LIN {X 0,Y 369.299,Z 673.807,A -85,B 0,C 180,E1 -13026.444,E2 -13026.444} C_VEL
LIN {X 0,Y 367.685,Z 686.752,A -85,B 0,C 180,E1 -13027.673,E2 -13027.673} C_VEL
LIN {X 0,Y 366.094,Z 698.777,A -85,B 0,C 180,E1 -13029.05,E2 -13029.05} C_VEL
LIN {X 0,Y 364.688,Z 709.985,A -85,B 0,C 180,E1 -13030.584,E2 -13030.584} C_VEL
LIN {X 0,Y 363.393,Z 720.355,A -85,B 0,C 180,E1 -13032.266,E2 -13032.266} C_VEL
LIN {X 0,Y 362.264,Z 730.519,A -85,B 0,C 180,E1 -13034.24,E2 -13034.24} C_VEL
LIN {X 0,Y 361.681,Z 737.904,A -85,B 0,C 180,E1 -13035.943,E2 -13035.943} C_VEL
LIN {X 0,Y 361.141,Z 746.082,A -85,B 0,C 180,E1 -13038.209,E2 -13038.209} C_VEL
LIN {X 0,Y 361.017,Z 752.615,A -85,B 0,C 180,E1 -13040.475,E2 -13040.475} C_VEL
LIN {X 0,Y 361.096,Z 756.535,A -85,B 0,C 180,E1 -13042.169,E2 -13042.169} C_VEL
LIN {X 0,Y 361.282,Z 760.576,A -85,B 0,C 180,E1 -13044.418,E2 -13044.418} C_VEL
LIN {X 0,Y 361.402,Z 762.102,A -85,B 0,C 180,E1 -13045.538,E2 -13045.538} C_VEL
LIN {X 0,Y 361.443,Z 764.123,A -85,B 0,C 180,E1 -13047.771,E2 -13047.771} C_VEL
LIN {X 0,Y 361.687,Z 764.698,A -85,B 0,C 180,E1 -13048.886,E2 -13048.886} C_VEL
LIN {X 0,Y 361.681,Z 764.869,A -85,B 0,C 180,E1 -13051.113,E2 -13051.113} C_VEL
LIN {X 0,Y 361.357,Z 763.796,A -85,B 0,C 180,E1 -13053.344,E2 -13053.344} C_VEL
LIN {X 0,Y 361.354,Z 762.831,A -85,B 0,C 180,E1 -13054.461,E2 -13054.461} C_VEL
LIN {X 0,Y 361.099,Z 759.485,A -85,B 0,C 180,E1 -13056.975,E2 -13056.975} C_VEL
LIN {X 0,Y 360.902,Z 754.467,A -85,B 0,C 180,E1 -13059.527,E2 -13059.527} C_VEL
LIN {X 0,Y 361.06,Z 748.6,A -85,B 0,C 180,E1 -13061.793,E2 -13061.793} C_VEL
LIN {X 0,Y 361.615,Z 741.459,A -85,B 0,C 180,E1 -13064.002,E2 -13064.002} C_VEL
LIN {X 0,Y 362.603,Z 732.201,A -85,B 0,C 180,E1 -13066.321,E2 -13066.321} C_VEL
LIN {X 0,Y 363.986,Z 722.704,A -85,B 0,C 180,E1 -13068.285,E2 -13068.285} C_VEL
LIN {X 0,Y 365.41,Z 713.269,A -85,B 0,C 180,E1 -13069.931,E2 -13069.931} C_VEL
LIN {X 0,Y 367.365,Z 700.79,A -85,B 0,C 180,E1 -13071.755,E2 -13071.755} C_VEL
LIN {X 0,Y 369.396,Z 688.323,A -85,B 0,C 180,E1 -13073.251,E2 -13073.251} C_VEL
LIN {X 0,Y 371.558,Z 674.683,A -85,B 0,C 180,E1 -13074.589,E2 -13074.589} C_VEL
LIN {X 0,Y 373.499,Z 661.351,A -85,B 0,C 180,E1 -13075.643,E2 -13075.643} C_VEL
LIN {X 0,Y 375.455,Z 646.833,A -85,B 0,C 180,E1 -13076.544,E2 -13076.544} C_VEL
LIN {X 0,Y 377.1,Z 631.865,A -85,B 0,C 180,E1 -13077.242,E2 -13077.242} C_VEL
LIN {X 0,Y 378.235,Z 616.394,A -85,B 0,C 180,E1 -13077.753,E2 -13077.753} C_VEL
LIN {X 0,Y 379.231,Z 585.25,A -85,B 0,C 180,E1 -13078.389,E2 -13078.389} C_VEL
LIN {X 0,Y 381.27,Z 506.213,A -85,B 0,C 180,E1 -13079.919,E2 -13079.919} C_VEL
LIN {X 0,Y 378.126,Z 480.693,A -85,B 0,C 180,E1 -13080.781,E2 -13080.781} C_VEL
LIN {X 0,Y 373.205,Z 450.4,A -85,B 0,C 180,E1 -13081.959,E2 -13081.959} C_VEL
LIN {X 0,Y 372.138,Z 444.262,A -85,B 0,C 180,E1 -13082.225,E2 -13082.225} C_VEL
LIN {X 0,Y 374.167,Z 428.518,A -85,B 0,C 180,E1 -13084.622,E2 -13084.622} C_VEL
LIN {X 0,Y 371.816,Z 418.27,A -85,B 0,C 180,E1 -13086.551,E2 -13086.551} C_VEL
LIN {X 0,Y 367.323,Z 402.801,A -85,B 0,C 180,E1 -13089.726,E2 -13089.726} C_VEL
LIN {X 0,Y 362.493,Z 388.181,A -85,B 0,C 180,E1 -13093.024,E2 -13093.024} C_VEL
LIN {X 0,Y 361.834,Z 386.038,A -85,B 0,C 180,E1 -13093.563,E2 -13093.563} C_VEL
LIN {X 0,Y 361.819,Z 386.036,A -85,B 0,C 180,E1 -13097.169,E2 -13097.169} C_VEL
LIN {X 0,Y 361.815,Z 386.035,A -85,B 0,C 180,E1 -13100.982,E2 -13100.982} C_VEL
LIN {X 0,Y 361.859,Z 386.036,A -85,B 0,C 180,E1 -13104.656,E2 -13104.656} C_VEL
LIN {X 0,Y 361.827,Z 386.041,A -85,B 0,C 180,E1 -13108.37,E2 -13108.37} C_VEL
LIN {X 0,Y 361.855,Z 386.038,A -85,B 0,C 180,E1 -13110.952,E2 -13110.952} C_VEL
LIN {X 0,Y 361.84,Z 386.038,A -85,B 0,C 180,E1 -13114.704,E2 -13114.704} C_VEL
LIN {X 0,Y 361.84,Z 386.037,A -85,B 0,C 180,E1 -13118.344,E2 -13118.344} C_VEL
LIN {X 0,Y 361.883,Z 386.031,A -85,B 0,C 180,E1 -13122.097,E2 -13122.097} C_VEL
LIN {X 0,Y 361.968,Z 386.018,A -85,B 0,C 180,E1 -13126.113,E2 -13126.113} C_VEL
LIN {X 0,Y 361.984,Z 386.013,A -85,B 0,C 180,E1 -13129.937,E2 -13129.937} C_VEL
LIN {X 0,Y 362.102,Z 385.997,A -85,B 0,C 180,E1 -13133.313,E2 -13133.313} C_VEL
LIN {X 0,Y 362.254,Z 385.977,A -85,B 0,C 180,E1 -13137.777,E2 -13137.777} C_VEL
LIN {X 0,Y 362.252,Z 385.981,A -85,B 0,C 180,E1 -13142.224,E2 -13142.224} C_VEL
LIN {X 0,Y 362.127,Z 385.971,A -85,B 0,C 180,E1 -13146.687,E2 -13146.687} C_VEL
LIN {X 0,Y 361.985,Z 386.016,A -85,B 0,C 180,E1 -13150.064,E2 -13150.064} C_VEL
LIN {X 0,Y 361.987,Z 385.994,A -85,B 0,C 180,E1 -13153.899,E2 -13153.899} C_VEL
LIN {X 0,Y 361.917,Z 386.026,A -85,B 0,C 180,E1 -13156.935,E2 -13156.935} C_VEL
LIN {X 0,Y 361.873,Z 386.012,A -85,B 0,C 180,E1 -13160.462,E2 -13160.462} C_VEL
LIN {X 0,Y 361.851,Z 386.036,A -85,B 0,C 180,E1 -13164.102,E2 -13164.102} C_VEL
LIN {X 0,Y 361.826,Z 386.029,A -85,B 0,C 180,E1 -13167.786,E2 -13167.786} C_VEL
LIN {X 0,Y 361.837,Z 386.026,A -85,B 0,C 180,E1 -13171.286,E2 -13171.286} C_VEL
LIN {X 0,Y 361.842,Z 386.04,A -85,B 0,C 180,E1 -13174.282,E2 -13174.282} C_VEL
LIN {X 0,Y 361.851,Z 386.028,A -85,B 0,C 180,E1 -13177.223,E2 -13177.223} C_VEL
LIN {X 0,Y 361.805,Z 386.033,A -85,B 0,C 180,E1 -13180.752,E2 -13180.752} C_VEL
LIN {X 0,Y 361.806,Z 386.032,A -85,B 0,C 180,E1 -13184.371,E2 -13184.371} C_VEL
LIN {X 0,Y 361.822,Z 386.054,A -85,B 0,C 180,E1 -13188.265,E2 -13188.265} C_VEL
LIN {X 0,Y 362.805,Z 388.821,A -85,B 0,C 180,E1 -13188.449,E2 -13188.449} C_VEL
LIN {X 0,Y 364.536,Z 391.406,A -85,B 0,C 180,E1 -13188.714,E2 -13188.714} C_VEL
LIN {X 0,Y 374.281,Z 407.605,A -85,B 0,C 180,E1 -13190.185,E2 -13190.185} C_VEL
LIN {X 0,Y 382.972,Z 423.782,A -85,B 0,C 180,E1 -13191.447,E2 -13191.447} C_VEL
LIN {X 0,Y 381.952,Z 465.159,A -85,B 0,C 180,E1 -13192.26,E2 -13192.26} C_VEL
LIN {X 0,Y 380.904,Z 509.738,A -85,B 0,C 180,E1 -13193.136,E2 -13193.136} C_VEL
LIN {X 0,Y 380.569,Z 526.045,A -85,B 0,C 180,E1 -13193.572,E2 -13193.572} C_VEL
LIN {X 0,Y 379.947,Z 539.867,A -85,B 0,C 180,E1 -13194.138,E2 -13194.138} C_VEL
LIN {X 0,Y 378.941,Z 553.918,A -85,B 0,C 180,E1 -13194.906,E2 -13194.906} C_VEL
LIN {X 0,Y 377.652,Z 567.962,A -85,B 0,C 180,E1 -13195.903,E2 -13195.903} C_VEL
LIN {X 0,Y 376.21,Z 580.784,A -85,B 0,C 180,E1 -13197.039,E2 -13197.039} C_VEL
LIN {X 0,Y 374.328,Z 593.837,A -85,B 0,C 180,E1 -13198.444,E2 -13198.444} C_VEL
LIN {X 0,Y 372.539,Z 605.519,A -85,B 0,C 180,E1 -13199.987,E2 -13199.987} C_VEL
LIN {X 0,Y 370.658,Z 616.335,A -85,B 0,C 180,E1 -13201.706,E2 -13201.706} C_VEL
LIN {X 0,Y 368.828,Z 626.128,A -85,B 0,C 180,E1 -13203.584,E2 -13203.584} C_VEL
LIN {X 0,Y 367.11,Z 635.125,A -85,B 0,C 180,E1 -13205.696,E2 -13205.696} C_VEL
LIN {X 0,Y 365.859,Z 641.208,A -85,B 0,C 180,E1 -13207.408,E2 -13207.408} C_VEL
LIN {X 0,Y 364.601,Z 647.773,A -85,B 0,C 180,E1 -13209.699,E2 -13209.699} C_VEL
LIN {X 0,Y 363.547,Z 652.854,A -85,B 0,C 180,E1 -13211.983,E2 -13211.983} C_VEL
LIN {X 0,Y 362.813,Z 656.581,A -85,B 0,C 180,E1 -13214.266,E2 -13214.266} C_VEL
LIN {X 0,Y 362.312,Z 659.044,A -85,B 0,C 180,E1 -13216.541,E2 -13216.541} C_VEL
LIN {X 0,Y 362.042,Z 660.342,A -85,B 0,C 180,E1 -13218.807,E2 -13218.807} C_VEL
LIN {X 0,Y 361.94,Z 660.526,A -85,B 0,C 180,E1 -13221.064,E2 -13221.064} C_VEL
LIN {X 0,Y 362.002,Z 659.615,A -85,B 0,C 180,E1 -13223.311,E2 -13223.311} C_VEL
LIN {X 0,Y 362.04,Z 657.636,A -85,B 0,C 180,E1 -13225.547,E2 -13225.547} C_VEL
LIN {X 0,Y 362.519,Z 654.445,A -85,B 0,C 180,E1 -13227.778,E2 -13227.778} C_VEL
LIN {X 0,Y 362.987,Z 650.057,A -85,B 0,C 180,E1 -13230,E2 -13230} C_VEL
LIN {X 0,Y 363.879,Z 644.327,A -85,B 0,C 180,E1 -13232.214,E2 -13232.214} C_VEL
LIN {X 0,Y 364.903,Z 637.153,A -85,B 0,C 180,E1 -13234.419,E2 -13234.419} C_VEL
LIN {X 0,Y 365.957,Z 629.485,A -85,B 0,C 180,E1 -13236.34,E2 -13236.34} C_VEL
LIN {X 0,Y 367.335,Z 620.266,A -85,B 0,C 180,E1 -13238.25,E2 -13238.25} C_VEL
LIN {X 0,Y 368.656,Z 610.885,A -85,B 0,C 180,E1 -13239.88,E2 -13239.88} C_VEL
LIN {X 0,Y 370.067,Z 599.768,A -85,B 0,C 180,E1 -13241.502,E2 -13241.502} C_VEL
LIN {X 0,Y 371.296,Z 588.808,A -85,B 0,C 180,E1 -13242.851,E2 -13242.851} C_VEL
LIN {X 0,Y 372.593,Z 576.994,A -85,B 0,C 180,E1 -13244.055,E2 -13244.055} C_VEL
LIN {X 0,Y 373.78,Z 564.26,A -85,B 0,C 180,E1 -13245.123,E2 -13245.123} C_VEL
LIN {X 0,Y 374.814,Z 551.249,A -85,B 0,C 180,E1 -13245.999,E2 -13245.999} C_VEL
LIN {X 0,Y 374.608,Z 545.819,A -85,B 0,C 180,E1 -13246.354,E2 -13246.354} C_VEL
LIN {X 0,Y 372.444,Z 537.038,A -85,B 0,C 180,E1 -13246.98,E2 -13246.98} C_VEL
LIN {X 0,Y 370.164,Z 528.099,A -85,B 0,C 180,E1 -13247.538,E2 -13247.538} C_VEL
LIN {X 0,Y 369.641,Z 522.425,A -85,B 0,C 180,E1 -13247.777,E2 -13247.777} C_VEL
LIN {X 0,Y 369.882,Z 504.154,A -85,B 0,C 180,E1 -13248.217,E2 -13248.217} C_VEL
LIN {X 0,Y 371.608,Z 421.809,A -85,B 0,C 180,E1 -13249.832,E2 -13249.832} C_VEL
LIN {X 0,Y 359.643,Z 396.831,A -85,B 0,C 180,E1 -13251.356,E2 -13251.356} C_VEL
LIN {X 0,Y 355.091,Z 388.184,A -85,B 0,C 180,E1 -13251.946,E2 -13251.946} C_VEL
LIN {X 0,Y 354.805,Z 386.914,A -85,B 0,C 180,E1 -13252.006,E2 -13252.006} C_VEL
LIN {X 0,Y 354.795,Z 386.917,A -85,B 0,C 180,E1 -13255.835,E2 -13255.835} C_VEL
LIN {X 0,Y 354.786,Z 386.9,A -85,B 0,C 180,E1 -13259.684,E2 -13259.684} C_VEL
LIN {X 0,Y 354.786,Z 386.917,A -85,B 0,C 180,E1 -13262.333,E2 -13262.333} C_VEL
LIN {X 0,Y 354.817,Z 386.911,A -85,B 0,C 180,E1 -13265.697,E2 -13265.697} C_VEL
LIN {X 0,Y 354.767,Z 386.914,A -85,B 0,C 180,E1 -13269.412,E2 -13269.412} C_VEL
LIN {X 0,Y 354.764,Z 386.918,A -85,B 0,C 180,E1 -13272.862,E2 -13272.862} C_VEL
LIN {X 0,Y 354.756,Z 386.918,A -85,B 0,C 180,E1 -13276.101,E2 -13276.101} C_VEL
LIN {X 0,Y 354.76,Z 386.921,A -85,B 0,C 180,E1 -13279.175,E2 -13279.175} C_VEL
LIN {X 0,Y 354.795,Z 386.91,A -85,B 0,C 180,E1 -13282.404,E2 -13282.404} C_VEL
LIN {X 0,Y 354.804,Z 386.916,A -85,B 0,C 180,E1 -13284.939,E2 -13284.939} C_VEL
LIN {X 0,Y 354.771,Z 386.918,A -85,B 0,C 180,E1 -13288.409,E2 -13288.409} C_VEL
LIN {X 0,Y 354.783,Z 386.913,A -85,B 0,C 180,E1 -13291.613,E2 -13291.613} C_VEL
LIN {X 0,Y 354.837,Z 386.903,A -85,B 0,C 180,E1 -13295.422,E2 -13295.422} C_VEL
LIN {X 0,Y 354.819,Z 386.914,A -85,B 0,C 180,E1 -13299.112,E2 -13299.112} C_VEL
LIN {X 0,Y 354.874,Z 386.901,A -85,B 0,C 180,E1 -13302.718,E2 -13302.718} C_VEL
LIN {X 0,Y 354.945,Z 386.884,A -85,B 0,C 180,E1 -13306.255,E2 -13306.255} C_VEL
LIN {X 0,Y 354.945,Z 386.856,A -85,B 0,C 180,E1 -13309.735,E2 -13309.735} C_VEL
LIN {X 0,Y 355.076,Z 386.874,A -85,B 0,C 180,E1 -13313.179,E2 -13313.179} C_VEL
LIN {X 0,Y 355.207,Z 386.852,A -85,B 0,C 180,E1 -13317.732,E2 -13317.732} C_VEL
LIN {X 0,Y 355.221,Z 386.855,A -85,B 0,C 180,E1 -13322.267,E2 -13322.267} C_VEL
LIN {X 0,Y 355.068,Z 386.878,A -85,B 0,C 180,E1 -13326.82,E2 -13326.82} C_VEL
LIN {X 0,Y 354.945,Z 386.892,A -85,B 0,C 180,E1 -13330.265,E2 -13330.265} C_VEL
LIN {X 0,Y 354.911,Z 386.892,A -85,B 0,C 180,E1 -13334.002,E2 -13334.002} C_VEL
LIN {X 0,Y 354.828,Z 386.905,A -85,B 0,C 180,E1 -13338.064,E2 -13338.064} C_VEL
LIN {X 0,Y 354.798,Z 386.91,A -85,B 0,C 180,E1 -13342.108,E2 -13342.108} C_VEL
LIN {X 0,Y 354.788,Z 386.913,A -85,B 0,C 180,E1 -13345.836,E2 -13345.836} C_VEL
LIN {X 0,Y 354.79,Z 386.914,A -85,B 0,C 180,E1 -13349.684,E2 -13349.684} C_VEL
LIN {X 0,Y 354.78,Z 386.911,A -85,B 0,C 180,E1 -13352.334,E2 -13352.334} C_VEL
LIN {X 0,Y 354.812,Z 386.914,A -85,B 0,C 180,E1 -13355.698,E2 -13355.698} C_VEL
LIN {X 0,Y 354.763,Z 386.911,A -85,B 0,C 180,E1 -13359.413,E2 -13359.413} C_VEL
LIN {X 0,Y 354.776,Z 386.91,A -85,B 0,C 180,E1 -13362.866,E2 -13362.866} C_VEL
LIN {X 0,Y 354.757,Z 386.916,A -85,B 0,C 180,E1 -13366.103,E2 -13366.103} C_VEL
LIN {X 0,Y 354.778,Z 386.916,A -85,B 0,C 180,E1 -13368.711,E2 -13368.711} C_VEL
LIN {X 0,Y 359.289,Z 402.611,A -85,B 0,C 180,E1 -13371.791,E2 -13371.791} C_VEL
LIN {X 0,Y 363.094,Z 417.355,A -85,B 0,C 180,E1 -13374.502,E2 -13374.502} C_VEL
LIN {X 0,Y 364.871,Z 425.465,A -85,B 0,C 180,E1 -13375.919,E2 -13375.919} C_VEL
LIN {X 0,Y 362.743,Z 445.555,A -85,B 0,C 180,E1 -13378.91,E2 -13378.91} C_VEL
LIN {X 0,Y 370.626,Z 506.012,A -85,B 0,C 180,E1 -13380.809,E2 -13380.809} C_VEL
LIN {X 0,Y 368.119,Z 614.078,A -85,B 0,C 180,E1 -13382.921,E2 -13382.921} C_VEL
LIN {X 0,Y 367.212,Z 629.994,A -85,B 0,C 180,E1 -13383.425,E2 -13383.425} C_VEL
LIN {X 0,Y 365.809,Z 645.847,A -85,B 0,C 180,E1 -13384.159,E2 -13384.159} C_VEL
LIN {X 0,Y 364.218,Z 659.938,A -85,B 0,C 180,E1 -13385.035,E2 -13385.035} C_VEL
LIN {X 0,Y 362.5,Z 673.746,A -85,B 0,C 180,E1 -13386.127,E2 -13386.127} C_VEL
LIN {X 0,Y 360.631,Z 687.834,A -85,B 0,C 180,E1 -13387.514,E2 -13387.514} C_VEL
LIN {X 0,Y 358.898,Z 700.613,A -85,B 0,C 180,E1 -13389.061,E2 -13389.061} C_VEL
LIN {X 0,Y 357.399,Z 711.936,A -85,B 0,C 180,E1 -13390.714,E2 -13390.714} C_VEL
LIN {X 0,Y 356.138,Z 722.116,A -85,B 0,C 180,E1 -13392.486,E2 -13392.486} C_VEL
LIN {X 0,Y 355.034,Z 731.814,A -85,B 0,C 180,E1 -13394.5,E2 -13394.5} C_VEL
LIN {X 0,Y 354.425,Z 739.831,A -85,B 0,C 180,E1 -13396.501,E2 -13396.501} C_VEL
LIN {X 0,Y 354.035,Z 746.652,A -85,B 0,C 180,E1 -13398.55,E2 -13398.55} C_VEL
LIN {X 0,Y 353.981,Z 752.856,A -85,B 0,C 180,E1 -13400.861,E2 -13400.861} C_VEL
LIN {X 0,Y 354.105,Z 757.614,A -85,B 0,C 180,E1 -13403.161,E2 -13403.161} C_VEL
LIN {X 0,Y 354.366,Z 761.025,A -85,B 0,C 180,E1 -13405.45,E2 -13405.45} C_VEL
LIN {X 0,Y 354.41,Z 763.069,A -85,B 0,C 180,E1 -13407.727,E2 -13407.727} C_VEL
LIN {X 0,Y 354.659,Z 763.66,A -85,B 0,C 180,E1 -13408.864,E2 -13408.864} C_VEL
LIN {X 0,Y 354.72,Z 763.919,A -85,B 0,C 180,E1 -13410,E2 -13410} C_VEL
LIN {X 0,Y 354.651,Z 763.859,A -85,B 0,C 180,E1 -13411.135,E2 -13411.135} C_VEL
LIN {X 0,Y 354.312,Z 762.81,A -85,B 0,C 180,E1 -13413.411,E2 -13413.411} C_VEL
LIN {X 0,Y 354.281,Z 761.854,A -85,B 0,C 180,E1 -13414.551,E2 -13414.551} C_VEL
LIN {X 0,Y 354.036,Z 758.733,A -85,B 0,C 180,E1 -13416.998,E2 -13416.998} C_VEL
LIN {X 0,Y 353.842,Z 754.793,A -85,B 0,C 180,E1 -13419.142,E2 -13419.142} C_VEL
LIN {X 0,Y 353.929,Z 749.283,A -85,B 0,C 180,E1 -13421.453,E2 -13421.453} C_VEL
LIN {X 0,Y 354.439,Z 742.344,A -85,B 0,C 180,E1 -13423.764,E2 -13423.764} C_VEL
LIN {X 0,Y 355.375,Z 733.796,A -85,B 0,C 180,E1 -13426.072,E2 -13426.072} C_VEL
LIN {X 0,Y 356.658,Z 724.783,A -85,B 0,C 180,E1 -13428.08,E2 -13428.08} C_VEL
LIN {X 0,Y 358.401,Z 714.051,A -85,B 0,C 180,E1 -13430.069,E2 -13430.069} C_VEL
LIN {X 0,Y 360.155,Z 703.126,A -85,B 0,C 180,E1 -13431.762,E2 -13431.762} C_VEL
LIN {X 0,Y 362.181,Z 691.322,A -85,B 0,C 180,E1 -13433.288,E2 -13433.288} C_VEL
LIN {X 0,Y 364.441,Z 678.552,A -85,B 0,C 180,E1 -13434.646,E2 -13434.646} C_VEL
LIN {X 0,Y 366.366,Z 665.859,A -85,B 0,C 180,E1 -13435.765,E2 -13435.765} C_VEL
LIN {X 0,Y 368.532,Z 651.258,A -85,B 0,C 180,E1 -13436.777,E2 -13436.777} C_VEL
LIN {X 0,Y 370.392,Z 635.923,A -85,B 0,C 180,E1 -13437.586,E2 -13437.586} C_VEL
LIN {X 0,Y 371.817,Z 620.699,A -85,B 0,C 180,E1 -13438.16,E2 -13438.16} C_VEL
LIN {X 0,Y 372.568,Z 604.883,A -85,B 0,C 180,E1 -13438.559,E2 -13438.559} C_VEL
LIN {X 0,Y 375.193,Z 506.281,A -85,B 0,C 180,E1 -13440.497,E2 -13440.497} C_VEL
LIN {X 0,Y 371.903,Z 480.176,A -85,B 0,C 180,E1 -13441.414,E2 -13441.414} C_VEL
LIN {X 0,Y 367.258,Z 451.386,A -85,B 0,C 180,E1 -13442.566,E2 -13442.566} C_VEL
LIN {X 0,Y 365.804,Z 443.045,A -85,B 0,C 180,E1 -13442.943,E2 -13442.943} C_VEL
LIN {X 0,Y 367.472,Z 430.974,A -85,B 0,C 180,E1 -13444.817,E2 -13444.817} C_VEL
LIN {X 0,Y 365.997,Z 423.398,A -85,B 0,C 180,E1 -13446.245,E2 -13446.245} C_VEL
LIN {X 0,Y 362.135,Z 409.596,A -85,B 0,C 180,E1 -13449.079,E2 -13449.079} C_VEL
LIN {X 0,Y 358.237,Z 397.221,A -85,B 0,C 180,E1 -13451.836,E2 -13451.836} C_VEL
LIN {X 0,Y 354.78,Z 386.904,A -85,B 0,C 180,E1 -13454.33,E2 -13454.33} C_VEL
LIN {X 0,Y 354.772,Z 386.918,A -85,B 0,C 180,E1 -13457.66,E2 -13457.66} C_VEL
LIN {X 0,Y 354.776,Z 386.913,A -85,B 0,C 180,E1 -13460.661,E2 -13460.661} C_VEL
LIN {X 0,Y 354.808,Z 386.911,A -85,B 0,C 180,E1 -13464.301,E2 -13464.301} C_VEL
LIN {X 0,Y 354.776,Z 386.918,A -85,B 0,C 180,E1 -13467.666,E2 -13467.666} C_VEL
LIN {X 0,Y 354.785,Z 386.919,A -85,B 0,C 180,E1 -13471.614,E2 -13471.614} C_VEL
LIN {X 0,Y 354.79,Z 386.913,A -85,B 0,C 180,E1 -13475.419,E2 -13475.419} C_VEL
LIN {X 0,Y 354.806,Z 386.909,A -85,B 0,C 180,E1 -13479.112,E2 -13479.112} C_VEL
LIN {X 0,Y 354.826,Z 386.908,A -85,B 0,C 180,E1 -13482.717,E2 -13482.717} C_VEL
LIN {X 0,Y 354.927,Z 386.894,A -85,B 0,C 180,E1 -13486.254,E2 -13486.254} C_VEL
LIN {X 0,Y 354.94,Z 386.891,A -85,B 0,C 180,E1 -13489.735,E2 -13489.735} C_VEL
LIN {X 0,Y 355.069,Z 386.873,A -85,B 0,C 180,E1 -13493.18,E2 -13493.18} C_VEL
LIN {X 0,Y 355.217,Z 386.853,A -85,B 0,C 180,E1 -13497.732,E2 -13497.732} C_VEL
LIN {X 0,Y 355.214,Z 386.858,A -85,B 0,C 180,E1 -13502.268,E2 -13502.268} C_VEL
LIN {X 0,Y 355.09,Z 386.846,A -85,B 0,C 180,E1 -13506.82,E2 -13506.82} C_VEL
LIN {X 0,Y 354.942,Z 386.895,A -85,B 0,C 180,E1 -13510.265,E2 -13510.265} C_VEL
LIN {X 0,Y 354.932,Z 386.871,A -85,B 0,C 180,E1 -13514.019,E2 -13514.019} C_VEL
LIN {X 0,Y 354.88,Z 386.904,A -85,B 0,C 180,E1 -13518.093,E2 -13518.093} C_VEL
LIN {X 0,Y 354.796,Z 386.901,A -85,B 0,C 180,E1 -13522.109,E2 -13522.109} C_VEL
LIN {X 0,Y 354.792,Z 386.903,A -85,B 0,C 180,E1 -13525.836,E2 -13525.836} C_VEL
LIN {X 0,Y 354.784,Z 386.918,A -85,B 0,C 180,E1 -13529.685,E2 -13529.685} C_VEL
LIN {X 0,Y 354.776,Z 386.902,A -85,B 0,C 180,E1 -13532.335,E2 -13532.335} C_VEL
LIN {X 0,Y 354.811,Z 386.909,A -85,B 0,C 180,E1 -13535.7,E2 -13535.7} C_VEL
LIN {X 0,Y 354.761,Z 386.917,A -85,B 0,C 180,E1 -13539.414,E2 -13539.414} C_VEL
LIN {X 0,Y 354.778,Z 386.915,A -85,B 0,C 180,E1 -13542.868,E2 -13542.868} C_VEL
LIN {X 0,Y 354.76,Z 386.918,A -85,B 0,C 180,E1 -13546.105,E2 -13546.105} C_VEL
LIN {X 0,Y 354.807,Z 387.079,A -85,B 0,C 180,E1 -13547.43,E2 -13547.43} C_VEL
LIN {X 0,Y 355.888,Z 389.917,A -85,B 0,C 180,E1 -13547.637,E2 -13547.637} C_VEL
LIN {X 0,Y 357.448,Z 392.028,A -85,B 0,C 180,E1 -13547.883,E2 -13547.883} C_VEL
LIN {X 0,Y 368.21,Z 409.846,A -85,B 0,C 180,E1 -13549.573,E2 -13549.573} C_VEL
LIN {X 0,Y 377.115,Z 426.325,A -85,B 0,C 180,E1 -13550.911,E2 -13550.911} C_VEL
LIN {X 0,Y 374.891,Z 509.395,A -85,B 0,C 180,E1 -13552.554,E2 -13552.554} C_VEL
LIN {X 0,Y 374.562,Z 526.103,A -85,B 0,C 180,E1 -13552.997,E2 -13552.997} C_VEL
LIN {X 0,Y 373.928,Z 539.875,A -85,B 0,C 180,E1 -13553.554,E2 -13553.554} C_VEL
LIN {X 0,Y 372.909,Z 553.763,A -85,B 0,C 180,E1 -13554.306,E2 -13554.306} C_VEL
LIN {X 0,Y 371.645,Z 567.491,A -85,B 0,C 180,E1 -13555.274,E2 -13555.274} C_VEL
LIN {X 0,Y 370.112,Z 580.607,A -85,B 0,C 180,E1 -13556.425,E2 -13556.425} C_VEL
LIN {X 0,Y 368.335,Z 592.698,A -85,B 0,C 180,E1 -13557.708,E2 -13557.708} C_VEL
LIN {X 0,Y 366.593,Z 603.892,A -85,B 0,C 180,E1 -13559.149,E2 -13559.149} C_VEL
LIN {X 0,Y 364.59,Z 615.061,A -85,B 0,C 180,E1 -13560.875,E2 -13560.875} C_VEL
LIN {X 0,Y 362.863,Z 624.3,A -85,B 0,C 180,E1 -13562.598,E2 -13562.598} C_VEL
LIN {X 0,Y 360.988,Z 633.438,A -85,B 0,C 180,E1 -13564.641,E2 -13564.641} C_VEL
LIN {X 0,Y 359.318,Z 641.377,A -85,B 0,C 180,E1 -13566.823,E2 -13566.823} C_VEL
LIN {X 0,Y 358.16,Z 646.951,A -85,B 0,C 180,E1 -13568.715,E2 -13568.715} C_VEL
LIN {X 0,Y 357.041,Z 652.123,A -85,B 0,C 180,E1 -13570.881,E2 -13570.881} C_VEL
LIN {X 0,Y 356.266,Z 655.706,A -85,B 0,C 180,E1 -13572.789,E2 -13572.789} C_VEL
LIN {X 0,Y 355.58,Z 658.841,A -85,B 0,C 180,E1 -13575.112,E2 -13575.112} C_VEL
LIN {X 0,Y 355.129,Z 660.782,A -85,B 0,C 180,E1 -13577.427,E2 -13577.427} C_VEL
LIN {X 0,Y 354.983,Z 661.574,A -85,B 0,C 180,E1 -13579.737,E2 -13579.737} C_VEL
LIN {X 0,Y 354.956,Z 661.272,A -85,B 0,C 180,E1 -13582.034,E2 -13582.034} C_VEL
LIN {X 0,Y 354.984,Z 659.896,A -85,B 0,C 180,E1 -13584.32,E2 -13584.32} C_VEL
LIN {X 0,Y 355.259,Z 657.361,A -85,B 0,C 180,E1 -13586.598,E2 -13586.598} C_VEL
LIN {X 0,Y 355.693,Z 653.639,A -85,B 0,C 180,E1 -13588.868,E2 -13588.868} C_VEL
LIN {X 0,Y 356.395,Z 648.667,A -85,B 0,C 180,E1 -13591.13,E2 -13591.13} C_VEL
LIN {X 0,Y 357.393,Z 642.313,A -85,B 0,C 180,E1 -13593.382,E2 -13593.382} C_VEL
LIN {X 0,Y 358.381,Z 635.495,A -85,B 0,C 180,E1 -13595.345,E2 -13595.345} C_VEL
LIN {X 0,Y 359.613,Z 627.3,A -85,B 0,C 180,E1 -13597.298,E2 -13597.298} C_VEL
LIN {X 0,Y 361.12,Z 617.434,A -85,B 0,C 180,E1 -13599.24,E2 -13599.24} C_VEL
LIN {X 0,Y 362.534,Z 607.375,A -85,B 0,C 180,E1 -13600.895,E2 -13600.895} C_VEL
LIN {X 0,Y 363.963,Z 595.362,A -85,B 0,C 180,E1 -13602.547,E2 -13602.547} C_VEL
LIN {X 0,Y 365.38,Z 583.311,A -85,B 0,C 180,E1 -13603.912,E2 -13603.912} C_VEL
LIN {X 0,Y 366.807,Z 570.113,A -85,B 0,C 180,E1 -13605.133,E2 -13605.133} C_VEL
LIN {X 0,Y 367.995,Z 556.465,A -85,B 0,C 180,E1 -13606.148,E2 -13606.148} C_VEL
LIN {X 0,Y 368.957,Z 542.058,A -85,B 0,C 180,E1 -13606.981,E2 -13606.981} C_VEL
LIN {X 0,Y 369.594,Z 526.392,A -85,B 0,C 180,E1 -13607.648,E2 -13607.648} C_VEL
LIN {X 0,Y 369.641,Z 522.425,A -85,B 0,C 180,E1 -13607.777,E2 -13607.777} C_VEL
LIN {X 0,Y 369.089,Z 518.601,A -85,B 0,C 180,E1 -13607.941,E2 -13607.941} C_VEL
LIN {X 0,Y 364.015,Z 506.797,A -85,B 0,C 180,E1 -13608.597,E2 -13608.597} C_VEL
LIN {X 0,Y 363.516,Z 502.934,A -85,B 0,C 180,E1 -13608.717,E2 -13608.717} C_VEL
LIN {X 0,Y 365.29,Z 423.859,A -85,B 0,C 180,E1 -13610.29,E2 -13610.29} C_VEL
LIN {X 0,Y 353.965,Z 400.322,A -85,B 0,C 180,E1 -13611.77,E2 -13611.77} C_VEL
LIN {X 0,Y 347.938,Z 388.774,A -85,B 0,C 180,E1 -13612.581,E2 -13612.581} C_VEL
LIN {X 0,Y 347.757,Z 387.829,A -85,B 0,C 180,E1 -13612.619,E2 -13612.619} C_VEL
LIN {X 0,Y 347.734,Z 387.796,A -85,B 0,C 180,E1 -13615.114,E2 -13615.114} C_VEL
LIN {X 0,Y 347.725,Z 387.799,A -85,B 0,C 180,E1 -13617.701,E2 -13617.701} C_VEL
LIN {X 0,Y 347.733,Z 387.778,A -85,B 0,C 180,E1 -13620.349,E2 -13620.349} C_VEL
LIN {X 0,Y 347.748,Z 387.789,A -85,B 0,C 180,E1 -13624.043,E2 -13624.043} C_VEL
LIN {X 0,Y 347.753,Z 387.79,A -85,B 0,C 180,E1 -13627.321,E2 -13627.321} C_VEL
LIN {X 0,Y 347.694,Z 387.792,A -85,B 0,C 180,E1 -13630.302,E2 -13630.302} C_VEL
LIN {X 0,Y 347.711,Z 387.792,A -85,B 0,C 180,E1 -13633.409,E2 -13633.409} C_VEL
LIN {X 0,Y 347.719,Z 387.796,A -85,B 0,C 180,E1 -13636.686,E2 -13636.686} C_VEL
LIN {X 0,Y 347.698,Z 387.798,A -85,B 0,C 180,E1 -13640.182,E2 -13640.182} C_VEL
LIN {X 0,Y 347.751,Z 387.788,A -85,B 0,C 180,E1 -13642.677,E2 -13642.677} C_VEL
LIN {X 0,Y 347.745,Z 387.784,A -85,B 0,C 180,E1 -13645.956,E2 -13645.956} C_VEL
LIN {X 0,Y 347.722,Z 387.794,A -85,B 0,C 180,E1 -13649.649,E2 -13649.649} C_VEL
LIN {X 0,Y 347.733,Z 387.796,A -85,B 0,C 180,E1 -13653.599,E2 -13653.599} C_VEL
LIN {X 0,Y 347.754,Z 387.783,A -85,B 0,C 180,E1 -13656.159,E2 -13656.159} C_VEL
LIN {X 0,Y 347.78,Z 387.783,A -85,B 0,C 180,E1 -13659.907,E2 -13659.907} C_VEL
LIN {X 0,Y 347.825,Z 387.786,A -85,B 0,C 180,E1 -13663.568,E2 -13663.568} C_VEL
LIN {X 0,Y 347.881,Z 387.752,A -85,B 0,C 180,E1 -13667.16,E2 -13667.16} C_VEL
LIN {X 0,Y 347.927,Z 387.741,A -85,B 0,C 180,E1 -13670.7,E2 -13670.7} C_VEL
LIN {X 0,Y 348.027,Z 387.757,A -85,B 0,C 180,E1 -13674.205,E2 -13674.205} C_VEL
LIN {X 0,Y 348.145,Z 387.731,A -85,B 0,C 180,E1 -13677.686,E2 -13677.686} C_VEL
LIN {X 0,Y 348.108,Z 387.748,A -85,B 0,C 180,E1 -13681.157,E2 -13681.157} C_VEL
LIN {X 0,Y 348.182,Z 387.732,A -85,B 0,C 180,E1 -13682.313,E2 -13682.313} C_VEL
LIN {X 0,Y 348.036,Z 387.755,A -85,B 0,C 180,E1 -13686.959,E2 -13686.959} C_VEL
LIN {X 0,Y 347.885,Z 387.771,A -85,B 0,C 180,E1 -13690.475,E2 -13690.475} C_VEL
LIN {X 0,Y 347.851,Z 387.771,A -85,B 0,C 180,E1 -13694.122,E2 -13694.122} C_VEL
LIN {X 0,Y 347.781,Z 387.782,A -85,B 0,C 180,E1 -13698.238,E2 -13698.238} C_VEL
LIN {X 0,Y 347.756,Z 387.793,A -85,B 0,C 180,E1 -13701.624,E2 -13701.624} C_VEL
LIN {X 0,Y 347.727,Z 387.795,A -85,B 0,C 180,E1 -13705.115,E2 -13705.115} C_VEL
LIN {X 0,Y 347.719,Z 387.798,A -85,B 0,C 180,E1 -13707.702,E2 -13707.702} C_VEL
LIN {X 0,Y 347.732,Z 387.796,A -85,B 0,C 180,E1 -13710.349,E2 -13710.349} C_VEL
LIN {X 0,Y 347.743,Z 387.781,A -85,B 0,C 180,E1 -13714.044,E2 -13714.044} C_VEL
LIN {X 0,Y 347.749,Z 387.791,A -85,B 0,C 180,E1 -13717.322,E2 -13717.322} C_VEL
LIN {X 0,Y 347.691,Z 387.802,A -85,B 0,C 180,E1 -13720.303,E2 -13720.303} C_VEL
LIN {X 0,Y 347.716,Z 387.794,A -85,B 0,C 180,E1 -13723.409,E2 -13723.409} C_VEL
LIN {X 0,Y 347.748,Z 387.793,A -85,B 0,C 180,E1 -13727.388,E2 -13727.388} C_VEL
LIN {X 0,Y 347.742,Z 387.828,A -85,B 0,C 180,E1 -13728.169,E2 -13728.169} C_VEL
LIN {X 0,Y 352.558,Z 404.527,A -85,B 0,C 180,E1 -13731.531,E2 -13731.531} C_VEL
LIN {X 0,Y 356.395,Z 419.51,A -85,B 0,C 180,E1 -13734.344,E2 -13734.344} C_VEL
LIN {X 0,Y 357.997,Z 426.146,A -85,B 0,C 180,E1 -13735.54,E2 -13735.54} C_VEL
LIN {X 0,Y 357.897,Z 429.124,A -85,B 0,C 180,E1 -13736.012,E2 -13736.012} C_VEL
LIN {X 0,Y 356.15,Z 444.378,A -85,B 0,C 180,E1 -13738.334,E2 -13738.334} C_VEL
LIN {X 0,Y 363.445,Z 500.474,A -85,B 0,C 180,E1 -13740.157,E2 -13740.157} C_VEL
LIN {X 0,Y 364.184,Z 506.791,A -85,B 0,C 180,E1 -13740.349,E2 -13740.349} C_VEL
LIN {X 0,Y 361.621,Z 613.533,A -85,B 0,C 180,E1 -13742.472,E2 -13742.472} C_VEL
LIN {X 0,Y 360.707,Z 629.283,A -85,B 0,C 180,E1 -13742.986,E2 -13742.986} C_VEL
LIN {X 0,Y 359.251,Z 645.039,A -85,B 0,C 180,E1 -13743.73,E2 -13743.73} C_VEL
LIN {X 0,Y 357.508,Z 659.907,A -85,B 0,C 180,E1 -13744.676,E2 -13744.676} C_VEL
LIN {X 0,Y 355.718,Z 673.665,A -85,B 0,C 180,E1 -13745.798,E2 -13745.798} C_VEL
LIN {X 0,Y 353.8,Z 687.566,A -85,B 0,C 180,E1 -13747.21,E2 -13747.21} C_VEL
LIN {X 0,Y 351.991,Z 700.214,A -85,B 0,C 180,E1 -13748.784,E2 -13748.784} C_VEL
LIN {X 0,Y 350.429,Z 711.609,A -85,B 0,C 180,E1 -13750.493,E2 -13750.493} C_VEL
LIN {X 0,Y 349.054,Z 722.32,A -85,B 0,C 180,E1 -13752.421,E2 -13752.421} C_VEL
LIN {X 0,Y 347.961,Z 731.818,A -85,B 0,C 180,E1 -13754.477,E2 -13754.477} C_VEL
LIN {X 0,Y 347.277,Z 740.138,A -85,B 0,C 180,E1 -13756.653,E2 -13756.653} C_VEL
LIN {X 0,Y 346.928,Z 747.164,A -85,B 0,C 180,E1 -13758.904,E2 -13758.904} C_VEL
LIN {X 0,Y 346.936,Z 753.026,A -85,B 0,C 180,E1 -13761.261,E2 -13761.261} C_VEL
LIN {X 0,Y 347.071,Z 756.507,A -85,B 0,C 180,E1 -13763.021,E2 -13763.021} C_VEL
LIN {X 0,Y 347.329,Z 759.942,A -85,B 0,C 180,E1 -13765.357,E2 -13765.357} C_VEL
LIN {X 0,Y 347.376,Z 762.015,A -85,B 0,C 180,E1 -13767.681,E2 -13767.681} C_VEL
LIN {X 0,Y 347.63,Z 762.621,A -85,B 0,C 180,E1 -13768.841,E2 -13768.841} C_VEL
LIN {X 0,Y 347.719,Z 762.899,A -85,B 0,C 180,E1 -13770,E2 -13770} C_VEL
LIN {X 0,Y 347.62,Z 762.849,A -85,B 0,C 180,E1 -13771.158,E2 -13771.158} C_VEL
LIN {X 0,Y 347.264,Z 761.826,A -85,B 0,C 180,E1 -13773.48,E2 -13773.48} C_VEL
LIN {X 0,Y 347.211,Z 760.88,A -85,B 0,C 180,E1 -13774.643,E2 -13774.643} C_VEL
LIN {X 0,Y 346.962,Z 757.978,A -85,B 0,C 180,E1 -13777.007,E2 -13777.007} C_VEL
LIN {X 0,Y 346.776,Z 753.857,A -85,B 0,C 180,E1 -13779.33,E2 -13779.33} C_VEL
LIN {X 0,Y 346.876,Z 748.378,A -85,B 0,C 180,E1 -13781.689,E2 -13781.689} C_VEL
LIN {X 0,Y 347.429,Z 741.474,A -85,B 0,C 180,E1 -13784.048,E2 -13784.048} C_VEL
LIN {X 0,Y 348.427,Z 732.969,A -85,B 0,C 180,E1 -13786.402,E2 -13786.402} C_VEL
LIN {X 0,Y 349.801,Z 724.009,A -85,B 0,C 180,E1 -13788.447,E2 -13788.447} C_VEL
LIN {X 0,Y 351.606,Z 713.333,A -85,B 0,C 180,E1 -13790.474,E2 -13790.474} C_VEL
LIN {X 0,Y 353.506,Z 702.489,A -85,B 0,C 180,E1 -13792.192,E2 -13792.192} C_VEL
LIN {X 0,Y 355.634,Z 690.778,A -85,B 0,C 180,E1 -13793.743,E2 -13793.743} C_VEL
LIN {X 0,Y 357.949,Z 678.119,A -85,B 0,C 180,E1 -13795.123,E2 -13795.123} C_VEL
LIN {X 0,Y 359.902,Z 665.955,A -85,B 0,C 180,E1 -13796.223,E2 -13796.223} C_VEL
LIN {X 0,Y 362.206,Z 651.136,A -85,B 0,C 180,E1 -13797.283,E2 -13797.283} C_VEL
LIN {X 0,Y 364.227,Z 635.425,A -85,B 0,C 180,E1 -13798.133,E2 -13798.133} C_VEL
LIN {X 0,Y 365.691,Z 620.437,A -85,B 0,C 180,E1 -13798.714,E2 -13798.714} C_VEL
LIN {X 0,Y 366.481,Z 605.097,A -85,B 0,C 180,E1 -13799.117,E2 -13799.117} C_VEL
LIN {X 0,Y 369.217,Z 507.346,A -85,B 0,C 180,E1 -13801.067,E2 -13801.067} C_VEL
LIN {X 0,Y 365.985,Z 481.321,A -85,B 0,C 180,E1 -13802.003,E2 -13802.003} C_VEL
LIN {X 0,Y 361.18,Z 451.219,A -85,B 0,C 180,E1 -13803.242,E2 -13803.242} C_VEL
LIN {X 0,Y 359.537,Z 441.924,A -85,B 0,C 180,E1 -13803.677,E2 -13803.677} C_VEL
LIN {X 0,Y 360.878,Z 432.771,A -85,B 0,C 180,E1 -13805.121,E2 -13805.121} C_VEL
LIN {X 0,Y 358.81,Z 423.379,A -85,B 0,C 180,E1 -13806.968,E2 -13806.968} C_VEL
LIN {X 0,Y 354.912,Z 409.677,A -85,B 0,C 180,E1 -13809.885,E2 -13809.885} C_VEL
LIN {X 0,Y 351.139,Z 397.807,A -85,B 0,C 180,E1 -13812.632,E2 -13812.632} C_VEL
LIN {X 0,Y 347.703,Z 387.776,A -85,B 0,C 180,E1 -13815.19,E2 -13815.19} C_VEL
LIN {X 0,Y 347.729,Z 387.791,A -85,B 0,C 180,E1 -13818.399,E2 -13818.399} C_VEL
LIN {X 0,Y 347.752,Z 387.79,A -85,B 0,C 180,E1 -13822.013,E2 -13822.013} C_VEL
LIN {X 0,Y 347.733,Z 387.796,A -85,B 0,C 180,E1 -13825.535,E2 -13825.535} C_VEL
LIN {X 0,Y 347.734,Z 387.797,A -85,B 0,C 180,E1 -13828.3,E2 -13828.3} C_VEL
LIN {X 0,Y 347.733,Z 387.798,A -85,B 0,C 180,E1 -13830.984,E2 -13830.984} C_VEL
LIN {X 0,Y 347.721,Z 387.797,A -85,B 0,C 180,E1 -13833.599,E2 -13833.599} C_VEL
LIN {X 0,Y 347.736,Z 387.792,A -85,B 0,C 180,E1 -13836.158,E2 -13836.158} C_VEL
LIN {X 0,Y 347.728,Z 387.793,A -85,B 0,C 180,E1 -13839.904,E2 -13839.904} C_VEL
LIN {X 0,Y 347.786,Z 387.785,A -85,B 0,C 180,E1 -13842.355,E2 -13842.355} C_VEL
LIN {X 0,Y 347.867,Z 387.774,A -85,B 0,C 180,E1 -13845.97,E2 -13845.97} C_VEL
LIN {X 0,Y 347.88,Z 387.771,A -85,B 0,C 180,E1 -13849.524,E2 -13849.524} C_VEL
LIN {X 0,Y 348.036,Z 387.75,A -85,B 0,C 180,E1 -13853.041,E2 -13853.041} C_VEL
LIN {X 0,Y 348.178,Z 387.73,A -85,B 0,C 180,E1 -13857.687,E2 -13857.687} C_VEL
LIN {X 0,Y 348.13,Z 387.737,A -85,B 0,C 180,E1 -13861.157,E2 -13861.157} C_VEL
LIN {X 0,Y 348.176,Z 387.735,A -85,B 0,C 180,E1 -13862.314,E2 -13862.314} C_VEL
LIN {X 0,Y 348.055,Z 387.721,A -85,B 0,C 180,E1 -13866.959,E2 -13866.959} C_VEL
LIN {X 0,Y 347.882,Z 387.776,A -85,B 0,C 180,E1 -13870.476,E2 -13870.476} C_VEL
LIN {X 0,Y 347.888,Z 387.747,A -85,B 0,C 180,E1 -13874.151,E2 -13874.151} C_VEL
LIN {X 0,Y 347.819,Z 387.784,A -85,B 0,C 180,E1 -13878.26,E2 -13878.26} C_VEL
LIN {X 0,Y 347.753,Z 387.771,A -85,B 0,C 180,E1 -13881.625,E2 -13881.625} C_VEL
LIN {X 0,Y 347.729,Z 387.788,A -85,B 0,C 180,E1 -13885.115,E2 -13885.115} C_VEL
LIN {X 0,Y 347.719,Z 387.783,A -85,B 0,C 180,E1 -13887.702,E2 -13887.702} C_VEL
LIN {X 0,Y 347.726,Z 387.796,A -85,B 0,C 180,E1 -13890.35,E2 -13890.35} C_VEL
LIN {X 0,Y 347.74,Z 387.796,A -85,B 0,C 180,E1 -13894.045,E2 -13894.045} C_VEL
LIN {X 0,Y 347.748,Z 387.784,A -85,B 0,C 180,E1 -13897.323,E2 -13897.323} C_VEL
LIN {X 0,Y 347.69,Z 387.791,A -85,B 0,C 180,E1 -13900.303,E2 -13900.303} C_VEL
LIN {X 0,Y 347.715,Z 387.788,A -85,B 0,C 180,E1 -13903.41,E2 -13903.41} C_VEL
LIN {X 0,Y 347.749,Z 387.984,A -85,B 0,C 180,E1 -13906.54,E2 -13906.54} C_VEL
LIN {X 0,Y 348.759,Z 390.683,A -85,B 0,C 180,E1 -13906.744,E2 -13906.744} C_VEL
LIN {X 0,Y 350.412,Z 392.859,A -85,B 0,C 180,E1 -13907.015,E2 -13907.015} C_VEL
LIN {X 0,Y 361.55,Z 411.052,A -85,B 0,C 180,E1 -13908.841,E2 -13908.841} C_VEL
LIN {X 0,Y 371.131,Z 428.607,A -85,B 0,C 180,E1 -13910.332,E2 -13910.332} C_VEL
LIN {X 0,Y 368.918,Z 510.327,A -85,B 0,C 180,E1 -13911.98,E2 -13911.98} C_VEL
LIN {X 0,Y 368.549,Z 527.38,A -85,B 0,C 180,E1 -13912.439,E2 -13912.439} C_VEL
LIN {X 0,Y 367.856,Z 541.519,A -85,B 0,C 180,E1 -13913.026,E2 -13913.026} C_VEL
LIN {X 0,Y 366.728,Z 555.895,A -85,B 0,C 180,E1 -13913.83,E2 -13913.83} C_VEL
LIN {X 0,Y 365.491,Z 568.839,A -85,B 0,C 180,E1 -13914.771,E2 -13914.771} C_VEL
LIN {X 0,Y 363.875,Z 581.885,A -85,B 0,C 180,E1 -13915.938,E2 -13915.938} C_VEL
LIN {X 0,Y 362.02,Z 593.924,A -85,B 0,C 180,E1 -13917.24,E2 -13917.24} C_VEL
LIN {X 0,Y 360.038,Z 606.066,A -85,B 0,C 180,E1 -13918.852,E2 -13918.852} C_VEL
LIN {X 0,Y 357.947,Z 617.039,A -85,B 0,C 180,E1 -13920.605,E2 -13920.605} C_VEL
LIN {X 0,Y 356.075,Z 626.513,A -85,B 0,C 180,E1 -13922.431,E2 -13922.431} C_VEL
LIN {X 0,Y 354.213,Z 635.157,A -85,B 0,C 180,E1 -13924.436,E2 -13924.436} C_VEL
LIN {X 0,Y 352.563,Z 642.48,A -85,B 0,C 180,E1 -13926.505,E2 -13926.505} C_VEL
LIN {X 0,Y 351.101,Z 649.222,A -85,B 0,C 180,E1 -13928.882,E2 -13928.882} C_VEL
LIN {X 0,Y 349.869,Z 654.436,A -85,B 0,C 180,E1 -13931.253,E2 -13931.253} C_VEL
LIN {X 0,Y 349.003,Z 658.271,A -85,B 0,C 180,E1 -13933.626,E2 -13933.626} C_VEL
LIN {X 0,Y 348.396,Z 660.863,A -85,B 0,C 180,E1 -13935.992,E2 -13935.992} C_VEL
LIN {X 0,Y 348.037,Z 662.292,A -85,B 0,C 180,E1 -13938.351,E2 -13938.351} C_VEL
LIN {X 0,Y 347.912,Z 662.6,A -85,B 0,C 180,E1 -13940.701,E2 -13940.701} C_VEL
LIN {X 0,Y 347.952,Z 661.816,A -85,B 0,C 180,E1 -13943.04,E2 -13943.04} C_VEL
LIN {X 0,Y 347.977,Z 659.929,A -85,B 0,C 180,E1 -13945.367,E2 -13945.367} C_VEL
LIN {X 0,Y 348.469,Z 656.837,A -85,B 0,C 180,E1 -13947.689,E2 -13947.689} C_VEL
LIN {X 0,Y 348.978,Z 652.583,A -85,B 0,C 180,E1 -13950,E2 -13950} C_VEL
LIN {X 0,Y 349.881,Z 647.007,A -85,B 0,C 180,E1 -13952.303,E2 -13952.303} C_VEL
LIN {X 0,Y 350.987,Z 639.988,A -85,B 0,C 180,E1 -13954.594,E2 -13954.594} C_VEL
LIN {X 0,Y 352.118,Z 632.496,A -85,B 0,C 180,E1 -13956.59,E2 -13956.59} C_VEL
LIN {X 0,Y 353.583,Z 623.478,A -85,B 0,C 180,E1 -13958.573,E2 -13958.573} C_VEL
LIN {X 0,Y 354.976,Z 614.338,A -85,B 0,C 180,E1 -13960.264,E2 -13960.264} C_VEL
LIN {X 0,Y 356.5,Z 603.491,A -85,B 0,C 180,E1 -13961.946,E2 -13961.946} C_VEL
LIN {X 0,Y 357.949,Z 591.619,A -85,B 0,C 180,E1 -13963.483,E2 -13963.483} C_VEL
LIN {X 0,Y 359.503,Z 578.532,A -85,B 0,C 180,E1 -13964.867,E2 -13964.867} C_VEL
LIN {X 0,Y 360.921,Z 563.917,A -85,B 0,C 180,E1 -13966.11,E2 -13966.11} C_VEL
LIN {X 0,Y 362.086,Z 549.361,A -85,B 0,C 180,E1 -13967.072,E2 -13967.072} C_VEL
LIN {X 0,Y 362.91,Z 534.098,A -85,B 0,C 180,E1 -13967.832,E2 -13967.832} C_VEL
LIN {X 0,Y 363.33,Z 519.356,A -85,B 0,C 180,E1 -13968.349,E2 -13968.349} C_VEL
LIN {X 0,Y 363.516,Z 502.934,A -85,B 0,C 180,E1 -13968.717,E2 -13968.717} C_VEL
LIN {X 0,Y 363.099,Z 497.131,A -85,B 0,C 180,E1 -13968.874,E2 -13968.874} C_VEL
LIN {X 0,Y 358.258,Z 478.519,A -85,B 0,C 180,E1 -13969.659,E2 -13969.659} C_VEL
LIN {X 0,Y 357.774,Z 472.717,A -85,B 0,C 180,E1 -13969.826,E2 -13969.826} C_VEL
LIN {X 0,Y 358.955,Z 425.963,A -85,B 0,C 180,E1 -13970.765,E2 -13970.765} C_VEL
LIN {X 0,Y 348.39,Z 403.939,A -85,B 0,C 180,E1 -13972.187,E2 -13972.187} C_VEL
LIN {X 0,Y 340.964,Z 389.815,A -85,B 0,C 180,E1 -13973.217,E2 -13973.217} C_VEL
LIN {X 0,Y 340.703,Z 388.671,A -85,B 0,C 180,E1 -13973.276,E2 -13973.276} C_VEL
LIN {X 0,Y 340.71,Z 388.671,A -85,B 0,C 180,E1 -13976.988,E2 -13976.988} C_VEL
LIN {X 0,Y 340.691,Z 388.661,A -85,B 0,C 180,E1 -13981.045,E2 -13981.045} C_VEL
LIN {X 0,Y 340.715,Z 388.672,A -85,B 0,C 180,E1 -13985.279,E2 -13985.279} C_VEL
LIN {X 0,Y 340.692,Z 388.671,A -85,B 0,C 180,E1 -13988.381,E2 -13988.381} C_VEL
LIN {X 0,Y 340.662,Z 388.674,A -85,B 0,C 180,E1 -13992.038,E2 -13992.038} C_VEL
LIN {X 0,Y 340.628,Z 388.682,A -85,B 0,C 180,E1 -13995.452,E2 -13995.452} C_VEL
LIN {X 0,Y 340.665,Z 388.672,A -85,B 0,C 180,E1 -13998.687,E2 -13998.687} C_VEL
LIN {X 0,Y 340.715,Z 388.663,A -85,B 0,C 180,E1 -14001.77,E2 -14001.77} C_VEL
LIN {X 0,Y 340.719,Z 388.662,A -85,B 0,C 180,E1 -14005.595,E2 -14005.595} C_VEL
LIN {X 0,Y 340.677,Z 388.676,A -85,B 0,C 180,E1 -14008.953,E2 -14008.953} C_VEL
LIN {X 0,Y 340.706,Z 388.67,A -85,B 0,C 180,E1 -14013.011,E2 -14013.011} C_VEL
LIN {X 0,Y 340.74,Z 388.658,A -85,B 0,C 180,E1 -14015.637,E2 -14015.637} C_VEL
LIN {X 0,Y 340.715,Z 388.667,A -85,B 0,C 180,E1 -14019.472,E2 -14019.472} C_VEL
LIN {X 0,Y 340.787,Z 388.656,A -85,B 0,C 180,E1 -14021.98,E2 -14021.98} C_VEL
LIN {X 0,Y 340.847,Z 388.643,A -85,B 0,C 180,E1 -14025.716,E2 -14025.716} C_VEL
LIN {X 0,Y 340.837,Z 388.61,A -85,B 0,C 180,E1 -14029.305,E2 -14029.305} C_VEL
LIN {X 0,Y 340.992,Z 388.626,A -85,B 0,C 180,E1 -14032.896,E2 -14032.896} C_VEL
LIN {X 0,Y 340.795,Z 388.661,A -85,B 0,C 180,E1 -14035.268,E2 -14035.268} C_VEL
LIN {X 0,Y 341.086,Z 388.61,A -85,B 0,C 180,E1 -14037.638,E2 -14037.638} C_VEL
LIN {X 0,Y 341.079,Z 388.623,A -85,B 0,C 180,E1 -14041.18,E2 -14041.18} C_VEL
LIN {X 0,Y 341.119,Z 388.612,A -85,B 0,C 180,E1 -14042.361,E2 -14042.361} C_VEL
LIN {X 0,Y 340.985,Z 388.634,A -85,B 0,C 180,E1 -14047.103,E2 -14047.103} C_VEL
LIN {X 0,Y 340.838,Z 388.649,A -85,B 0,C 180,E1 -14050.695,E2 -14050.695} C_VEL
LIN {X 0,Y 340.806,Z 388.648,A -85,B 0,C 180,E1 -14054.327,E2 -14054.327} C_VEL
LIN {X 0,Y 340.744,Z 388.658,A -85,B 0,C 180,E1 -14058.422,E2 -14058.422} C_VEL
LIN {X 0,Y 340.712,Z 388.667,A -85,B 0,C 180,E1 -14061.842,E2 -14061.842} C_VEL
LIN {X 0,Y 340.661,Z 388.674,A -85,B 0,C 180,E1 -14065.673,E2 -14065.673} C_VEL
LIN {X 0,Y 340.67,Z 388.674,A -85,B 0,C 180,E1 -14068.326,E2 -14068.326} C_VEL
LIN {X 0,Y 340.687,Z 388.673,A -85,B 0,C 180,E1 -14071.045,E2 -14071.045} C_VEL
LIN {X 0,Y 340.709,Z 388.667,A -85,B 0,C 180,E1 -14075.28,E2 -14075.28} C_VEL
LIN {X 0,Y 340.687,Z 388.66,A -85,B 0,C 180,E1 -14078.382,E2 -14078.382} C_VEL
LIN {X 0,Y 340.685,Z 388.664,A -85,B 0,C 180,E1 -14082.044,E2 -14082.044} C_VEL
LIN {X 0,Y 340.645,Z 388.674,A -85,B 0,C 180,E1 -14086.228,E2 -14086.228} C_VEL
LIN {X 0,Y 340.721,Z 388.669,A -85,B 0,C 180,E1 -14087.59,E2 -14087.59} C_VEL
LIN {X 0,Y 345.081,Z 403.648,A -85,B 0,C 180,E1 -14090.707,E2 -14090.707} C_VEL
LIN {X 0,Y 349.301,Z 419.911,A -85,B 0,C 180,E1 -14093.86,E2 -14093.86} C_VEL
LIN {X 0,Y 351.28,Z 428.81,A -85,B 0,C 180,E1 -14095.489,E2 -14095.489} C_VEL
LIN {X 0,Y 349.555,Z 443.638,A -85,B 0,C 180,E1 -14097.762,E2 -14097.762} C_VEL
LIN {X 0,Y 355.495,Z 488.791,A -85,B 0,C 180,E1 -14099.278,E2 -14099.278} C_VEL
LIN {X 0,Y 357.795,Z 507.812,A -85,B 0,C 180,E1 -14099.88,E2 -14099.88} C_VEL
LIN {X 0,Y 355.151,Z 612.913,A -85,B 0,C 180,E1 -14102.007,E2 -14102.007} C_VEL
LIN {X 0,Y 354.205,Z 628.508,A -85,B 0,C 180,E1 -14102.528,E2 -14102.528} C_VEL
LIN {X 0,Y 352.699,Z 644.183,A -85,B 0,C 180,E1 -14103.283,E2 -14103.283} C_VEL
LIN {X 0,Y 351.046,Z 657.402,A -85,B 0,C 180,E1 -14104.127,E2 -14104.127} C_VEL
LIN {X 0,Y 349.408,Z 670.347,A -85,B 0,C 180,E1 -14105.173,E2 -14105.173} C_VEL
LIN {X 0,Y 347.589,Z 683.366,A -85,B 0,C 180,E1 -14106.464,E2 -14106.464} C_VEL
LIN {X 0,Y 345.792,Z 695.449,A -85,B 0,C 180,E1 -14107.914,E2 -14107.914} C_VEL
LIN {X 0,Y 344.297,Z 705.777,A -85,B 0,C 180,E1 -14109.383,E2 -14109.383} C_VEL
LIN {X 0,Y 342.811,Z 716.332,A -85,B 0,C 180,E1 -14111.162,E2 -14111.162} C_VEL
LIN {X 0,Y 341.445,Z 726.658,A -85,B 0,C 180,E1 -14113.252,E2 -14113.252} C_VEL
LIN {X 0,Y 340.608,Z 735.292,A -85,B 0,C 180,E1 -14115.359,E2 -14115.359} C_VEL
LIN {X 0,Y 340.017,Z 742.439,A -85,B 0,C 180,E1 -14117.465,E2 -14117.465} C_VEL
LIN {X 0,Y 339.838,Z 749.106,A -85,B 0,C 180,E1 -14119.876,E2 -14119.876} C_VEL
LIN {X 0,Y 339.952,Z 754.395,A -85,B 0,C 180,E1 -14122.337,E2 -14122.337} C_VEL
LIN {X 0,Y 340.099,Z 757.289,A -85,B 0,C 180,E1 -14124.069,E2 -14124.069} C_VEL
LIN {X 0,Y 340.291,Z 758.853,A -85,B 0,C 180,E1 -14125.261,E2 -14125.261} C_VEL
LIN {X 0,Y 340.341,Z 760.959,A -85,B 0,C 180,E1 -14127.633,E2 -14127.633} C_VEL
LIN {X 0,Y 340.601,Z 761.582,A -85,B 0,C 180,E1 -14128.817,E2 -14128.817} C_VEL
LIN {X 0,Y 340.714,Z 761.879,A -85,B 0,C 180,E1 -14130,E2 -14130} C_VEL
LIN {X 0,Y 340.589,Z 761.839,A -85,B 0,C 180,E1 -14131.182,E2 -14131.182} C_VEL
LIN {X 0,Y 340.216,Z 760.842,A -85,B 0,C 180,E1 -14133.552,E2 -14133.552} C_VEL
LIN {X 0,Y 340.144,Z 759.907,A -85,B 0,C 180,E1 -14134.74,E2 -14134.74} C_VEL
LIN {X 0,Y 339.879,Z 757.051,A -85,B 0,C 180,E1 -14137.126,E2 -14137.126} C_VEL
LIN {X 0,Y 339.689,Z 752.92,A -85,B 0,C 180,E1 -14139.526,E2 -14139.526} C_VEL
LIN {X 0,Y 339.828,Z 747.476,A -85,B 0,C 180,E1 -14141.935,E2 -14141.935} C_VEL
LIN {X 0,Y 340.453,Z 740.613,A -85,B 0,C 180,E1 -14144.342,E2 -14144.342} C_VEL
LIN {X 0,Y 341.475,Z 732.147,A -85,B 0,C 180,E1 -14146.746,E2 -14146.746} C_VEL
LIN {X 0,Y 342.991,Z 723.249,A -85,B 0,C 180,E1 -14148.827,E2 -14148.827} C_VEL
LIN {X 0,Y 344.858,Z 712.632,A -85,B 0,C 180,E1 -14150.893,E2 -14150.893} C_VEL
LIN {X 0,Y 346.873,Z 701.86,A -85,B 0,C 180,E1 -14152.64,E2 -14152.64} C_VEL
LIN {X 0,Y 349.101,Z 690.236,A -85,B 0,C 180,E1 -14154.215,E2 -14154.215} C_VEL
LIN {X 0,Y 351.491,Z 677.686,A -85,B 0,C 180,E1 -14155.618,E2 -14155.618} C_VEL
LIN {X 0,Y 353.732,Z 664.353,A -85,B 0,C 180,E1 -14156.839,E2 -14156.839} C_VEL
LIN {X 0,Y 356.072,Z 649.947,A -85,B 0,C 180,E1 -14157.873,E2 -14157.873} C_VEL
LIN {X 0,Y 358.183,Z 634.181,A -85,B 0,C 180,E1 -14158.731,E2 -14158.731} C_VEL
LIN {X 0,Y 359.642,Z 619.138,A -85,B 0,C 180,E1 -14159.324,E2 -14159.324} C_VEL
LIN {X 0,Y 360.488,Z 603.663,A -85,B 0,C 180,E1 -14159.729,E2 -14159.729} C_VEL
LIN {X 0,Y 363.294,Z 508.253,A -85,B 0,C 180,E1 -14161.659,E2 -14161.659} C_VEL
LIN {X 0,Y 360.091,Z 482.297,A -85,B 0,C 180,E1 -14162.619,E2 -14162.619} C_VEL
LIN {X 0,Y 355.969,Z 455.874,A -85,B 0,C 180,E1 -14163.728,E2 -14163.728} C_VEL
LIN {X 0,Y 353.324,Z 440.71,A -85,B 0,C 180,E1 -14164.448,E2 -14164.448} C_VEL
LIN {X 0,Y 354.195,Z 433.936,A -85,B 0,C 180,E1 -14165.558,E2 -14165.558} C_VEL
LIN {X 0,Y 351.941,Z 424.636,A -85,B 0,C 180,E1 -14167.461,E2 -14167.461} C_VEL
LIN {X 0,Y 348.214,Z 411.502,A -85,B 0,C 180,E1 -14170.332,E2 -14170.332} C_VEL
LIN {X 0,Y 343.999,Z 398.249,A -85,B 0,C 180,E1 -14173.509,E2 -14173.509} C_VEL
LIN {X 0,Y 340.66,Z 388.654,A -85,B 0,C 180,E1 -14176.052,E2 -14176.052} C_VEL
LIN {X 0,Y 340.659,Z 388.67,A -85,B 0,C 180,E1 -14178.687,E2 -14178.687} C_VEL
LIN {X 0,Y 340.708,Z 388.665,A -85,B 0,C 180,E1 -14181.77,E2 -14181.77} C_VEL
LIN {X 0,Y 340.712,Z 388.671,A -85,B 0,C 180,E1 -14185.595,E2 -14185.595} C_VEL
LIN {X 0,Y 340.683,Z 388.67,A -85,B 0,C 180,E1 -14188.954,E2 -14188.954} C_VEL
LIN {X 0,Y 340.698,Z 388.67,A -85,B 0,C 180,E1 -14193.011,E2 -14193.011} C_VEL
LIN {X 0,Y 340.688,Z 388.676,A -85,B 0,C 180,E1 -14196.925,E2 -14196.925} C_VEL
LIN {X 0,Y 340.678,Z 388.678,A -85,B 0,C 180,E1 -14200.727,E2 -14200.727} C_VEL
LIN {X 0,Y 340.716,Z 388.667,A -85,B 0,C 180,E1 -14203.215,E2 -14203.215} C_VEL
LIN {X 0,Y 340.824,Z 388.653,A -85,B 0,C 180,E1 -14206.89,E2 -14206.89} C_VEL
LIN {X 0,Y 340.868,Z 388.645,A -85,B 0,C 180,E1 -14210.506,E2 -14210.506} C_VEL
LIN {X 0,Y 340.985,Z 388.629,A -85,B 0,C 180,E1 -14212.897,E2 -14212.897} C_VEL
LIN {X 0,Y 340.803,Z 388.658,A -85,B 0,C 180,E1 -14215.269,E2 -14215.269} C_VEL
LIN {X 0,Y 341.116,Z 388.61,A -85,B 0,C 180,E1 -14217.639,E2 -14217.639} C_VEL
LIN {X 0,Y 341.099,Z 388.613,A -85,B 0,C 180,E1 -14221.181,E2 -14221.181} C_VEL
LIN {X 0,Y 341.114,Z 388.615,A -85,B 0,C 180,E1 -14222.362,E2 -14222.362} C_VEL
LIN {X 0,Y 340.988,Z 388.601,A -85,B 0,C 180,E1 -14226.713,E2 -14226.713} C_VEL
LIN {X 0,Y 340.869,Z 388.645,A -85,B 0,C 180,E1 -14229.494,E2 -14229.494} C_VEL
LIN {X 0,Y 340.832,Z 388.635,A -85,B 0,C 180,E1 -14233.11,E2 -14233.11} C_VEL
LIN {X 0,Y 340.764,Z 388.658,A -85,B 0,C 180,E1 -14236.783,E2 -14236.783} C_VEL
LIN {X 0,Y 340.747,Z 388.654,A -85,B 0,C 180,E1 -14239.269,E2 -14239.269} C_VEL
LIN {X 0,Y 340.69,Z 388.668,A -85,B 0,C 180,E1 -14243.076,E2 -14243.076} C_VEL
LIN {X 0,Y 340.701,Z 388.651,A -85,B 0,C 180,E1 -14246.989,E2 -14246.989} C_VEL
LIN {X 0,Y 340.682,Z 388.663,A -85,B 0,C 180,E1 -14251.047,E2 -14251.047} C_VEL
LIN {X 0,Y 340.708,Z 388.669,A -85,B 0,C 180,E1 -14255.281,E2 -14255.281} C_VEL
LIN {X 0,Y 340.686,Z 388.674,A -85,B 0,C 180,E1 -14258.384,E2 -14258.384} C_VEL
LIN {X 0,Y 340.687,Z 388.673,A -85,B 0,C 180,E1 -14262.046,E2 -14262.046} C_VEL
LIN {X 0,Y 340.686,Z 388.806,A -85,B 0,C 180,E1 -14265.599,E2 -14265.599} C_VEL
LIN {X 0,Y 341.677,Z 391.547,A -85,B 0,C 180,E1 -14265.811,E2 -14265.811} C_VEL
LIN {X 0,Y 343.45,Z 393.862,A -85,B 0,C 180,E1 -14266.116,E2 -14266.116} C_VEL
LIN {X 0,Y 353.167,Z 409.414,A -85,B 0,C 180,E1 -14267.787,E2 -14267.787} C_VEL
LIN {X 0,Y 361.764,Z 424.395,A -85,B 0,C 180,E1 -14269.189,E2 -14269.189} C_VEL
LIN {X 0,Y 365.309,Z 431.072,A -85,B 0,C 180,E1 -14269.751,E2 -14269.751} C_VEL
LIN {X 0,Y 362.985,Z 510.365,A -85,B 0,C 180,E1 -14271.366,E2 -14271.366} C_VEL
LIN {X 0,Y 362.628,Z 527.505,A -85,B 0,C 180,E1 -14271.827,E2 -14271.827} C_VEL
LIN {X 0,Y 361.92,Z 541.714,A -85,B 0,C 180,E1 -14272.411,E2 -14272.411} C_VEL
LIN {X 0,Y 360.733,Z 556.39,A -85,B 0,C 180,E1 -14273.233,E2 -14273.233} C_VEL
LIN {X 0,Y 359.346,Z 570.201,A -85,B 0,C 180,E1 -14274.249,E2 -14274.249} C_VEL
LIN {X 0,Y 357.719,Z 582.755,A -85,B 0,C 180,E1 -14275.389,E2 -14275.389} C_VEL
LIN {X 0,Y 355.726,Z 595.173,A -85,B 0,C 180,E1 -14276.754,E2 -14276.754} C_VEL
LIN {X 0,Y 353.852,Z 606.292,A -85,B 0,C 180,E1 -14278.244,E2 -14278.244} C_VEL
LIN {X 0,Y 351.649,Z 617.398,A -85,B 0,C 180,E1 -14280.025,E2 -14280.025} C_VEL
LIN {X 0,Y 349.675,Z 626.97,A -85,B 0,C 180,E1 -14281.882,E2 -14281.882} C_VEL
LIN {X 0,Y 347.674,Z 635.695,A -85,B 0,C 180,E1 -14283.919,E2 -14283.919} C_VEL
LIN {X 0,Y 345.875,Z 643.39,A -85,B 0,C 180,E1 -14286.118,E2 -14286.118} C_VEL
LIN {X 0,Y 344.357,Z 649.922,A -85,B 0,C 180,E1 -14288.448,E2 -14288.448} C_VEL
LIN {X 0,Y 343.059,Z 655.21,A -85,B 0,C 180,E1 -14290.867,E2 -14290.867} C_VEL
LIN {X 0,Y 342.116,Z 659.117,A -85,B 0,C 180,E1 -14293.287,E2 -14293.287} C_VEL
LIN {X 0,Y 341.454,Z 661.775,A -85,B 0,C 180,E1 -14295.701,E2 -14295.701} C_VEL
LIN {X 0,Y 341.037,Z 663.27,A -85,B 0,C 180,E1 -14298.108,E2 -14298.108} C_VEL
LIN {X 0,Y 340.899,Z 663.638,A -85,B 0,C 180,E1 -14300.508,E2 -14300.508} C_VEL
LIN {X 0,Y 340.928,Z 662.907,A -85,B 0,C 180,E1 -14302.896,E2 -14302.896} C_VEL
LIN {X 0,Y 340.943,Z 661.057,A -85,B 0,C 180,E1 -14305.271,E2 -14305.271} C_VEL
LIN {X 0,Y 341.442,Z 658.03,A -85,B 0,C 180,E1 -14307.641,E2 -14307.641} C_VEL
LIN {X 0,Y 341.968,Z 653.843,A -85,B 0,C 180,E1 -14310,E2 -14310} C_VEL
LIN {X 0,Y 342.877,Z 648.341,A -85,B 0,C 180,E1 -14312.35,E2 -14312.35} C_VEL
LIN {X 0,Y 344.018,Z 641.401,A -85,B 0,C 180,E1 -14314.688,E2 -14314.688} C_VEL
LIN {X 0,Y 345.384,Z 632.806,A -85,B 0,C 180,E1 -14317.013,E2 -14317.013} C_VEL
LIN {X 0,Y 346.923,Z 623.644,A -85,B 0,C 180,E1 -14319.033,E2 -14319.033} C_VEL
LIN {X 0,Y 348.391,Z 614.334,A -85,B 0,C 180,E1 -14320.754,E2 -14320.754} C_VEL
LIN {X 0,Y 349.949,Z 603.307,A -85,B 0,C 180,E1 -14322.468,E2 -14322.468} C_VEL
LIN {X 0,Y 351.369,Z 592.423,A -85,B 0,C 180,E1 -14323.888,E2 -14323.888} C_VEL
LIN {X 0,Y 352.968,Z 579.295,A -85,B 0,C 180,E1 -14325.297,E2 -14325.297} C_VEL
LIN {X 0,Y 354.263,Z 566.416,A -85,B 0,C 180,E1 -14326.421,E2 -14326.421} C_VEL
LIN {X 0,Y 355.481,Z 552.279,A -85,B 0,C 180,E1 -14327.399,E2 -14327.399} C_VEL
LIN {X 0,Y 356.369,Z 537.715,A -85,B 0,C 180,E1 -14328.17,E2 -14328.17} C_VEL
LIN {X 0,Y 356.842,Z 522.505,A -85,B 0,C 180,E1 -14328.75,E2 -14328.75} C_VEL
LIN {X 0,Y 357.226,Z 496.153,A -85,B 0,C 180,E1 -14329.352,E2 -14329.352} C_VEL
LIN {X 0,Y 357.774,Z 472.717,A -85,B 0,C 180,E1 -14329.826,E2 -14329.826} C_VEL
LIN {X 0,Y 357.315,Z 466.913,A -85,B 0,C 180,E1 -14329.991,E2 -14329.991} C_VEL
LIN {X 0,Y 352.724,Z 448.258,A -85,B 0,C 180,E1 -14330.791,E2 -14330.791} C_VEL
LIN {X 0,Y 352.333,Z 442.453,A -85,B 0,C 180,E1 -14330.956,E2 -14330.956} C_VEL
LIN {X 0,Y 352.583,Z 427.844,A -85,B 0,C 180,E1 -14331.266,E2 -14331.266} C_VEL
LIN {X 0,Y 342.341,Z 406.566,A -85,B 0,C 180,E1 -14332.686,E2 -14332.686} C_VEL
LIN {X 0,Y 333.884,Z 390.575,A -85,B 0,C 180,E1 -14333.899,E2 -14333.899} C_VEL
LIN {X 0,Y 333.668,Z 389.549,A -85,B 0,C 180,E1 -14333.971,E2 -14333.971} C_VEL
LIN {X 0,Y 333.643,Z 389.553,A -85,B 0,C 180,E1 -14337.784,E2 -14337.784} C_VEL
LIN {X 0,Y 333.655,Z 389.531,A -85,B 0,C 180,E1 -14340.366,E2 -14340.366} C_VEL
LIN {X 0,Y 333.635,Z 389.55,A -85,B 0,C 180,E1 -14343.208,E2 -14343.208} C_VEL
LIN {X 0,Y 333.672,Z 389.544,A -85,B 0,C 180,E1 -14346.139,E2 -14346.139} C_VEL
LIN {X 0,Y 333.618,Z 389.55,A -85,B 0,C 180,E1 -14349.196,E2 -14349.196} C_VEL
LIN {X 0,Y 333.606,Z 389.554,A -85,B 0,C 180,E1 -14352.494,E2 -14352.494} C_VEL
LIN {X 0,Y 333.587,Z 389.556,A -85,B 0,C 180,E1 -14355.953,E2 -14355.953} C_VEL
LIN {X 0,Y 333.599,Z 389.559,A -85,B 0,C 180,E1 -14359.324,E2 -14359.324} C_VEL
LIN {X 0,Y 333.658,Z 389.548,A -85,B 0,C 180,E1 -14363.168,E2 -14363.168} C_VEL
LIN {X 0,Y 333.669,Z 389.542,A -85,B 0,C 180,E1 -14365.34,E2 -14365.34} C_VEL
LIN {X 0,Y 333.615,Z 389.553,A -85,B 0,C 180,E1 -14368.22,E2 -14368.22} C_VEL
LIN {X 0,Y 333.619,Z 389.546,A -85,B 0,C 180,E1 -14371.019,E2 -14371.019} C_VEL
LIN {X 0,Y 333.692,Z 389.54,A -85,B 0,C 180,E1 -14375.088,E2 -14375.088} C_VEL
LIN {X 0,Y 333.653,Z 389.55,A -85,B 0,C 180,E1 -14379.017,E2 -14379.017} C_VEL
LIN {X 0,Y 333.735,Z 389.531,A -85,B 0,C 180,E1 -14381.586,E2 -14381.586} C_VEL
LIN {X 0,Y 333.803,Z 389.522,A -85,B 0,C 180,E1 -14385.576,E2 -14385.576} C_VEL
LIN {X 0,Y 333.808,Z 389.484,A -85,B 0,C 180,E1 -14389.077,E2 -14389.077} C_VEL
LIN {X 0,Y 333.948,Z 389.502,A -85,B 0,C 180,E1 -14392.745,E2 -14392.745} C_VEL
LIN {X 0,Y 333.763,Z 389.536,A -85,B 0,C 180,E1 -14395.168,E2 -14395.168} C_VEL
LIN {X 0,Y 334.029,Z 389.489,A -85,B 0,C 180,E1 -14397.588,E2 -14397.588} C_VEL
LIN {X 0,Y 334.05,Z 389.499,A -85,B 0,C 180,E1 -14401.205,E2 -14401.205} C_VEL
LIN {X 0,Y 334.06,Z 389.491,A -85,B 0,C 180,E1 -14402.411,E2 -14402.411} C_VEL
LIN {X 0,Y 333.973,Z 389.508,A -85,B 0,C 180,E1 -14406.039,E2 -14406.039} C_VEL
LIN {X 0,Y 333.907,Z 389.508,A -85,B 0,C 180,E1 -14408.472,E2 -14408.472} C_VEL
LIN {X 0,Y 333.779,Z 389.532,A -85,B 0,C 180,E1 -14412.155,E2 -14412.155} C_VEL
LIN {X 0,Y 333.728,Z 389.53,A -85,B 0,C 180,E1 -14414.638,E2 -14414.638} C_VEL
LIN {X 0,Y 333.683,Z 389.537,A -85,B 0,C 180,E1 -14418.6,E2 -14418.6} C_VEL
LIN {X 0,Y 333.642,Z 389.544,A -85,B 0,C 180,E1 -14422.281,E2 -14422.281} C_VEL
LIN {X 0,Y 333.649,Z 389.549,A -85,B 0,C 180,E1 -14425.077,E2 -14425.077} C_VEL
LIN {X 0,Y 333.624,Z 389.551,A -85,B 0,C 180,E1 -14428.98,E2 -14428.98} C_VEL
LIN {X 0,Y 333.638,Z 389.544,A -85,B 0,C 180,E1 -14432.587,E2 -14432.587} C_VEL
LIN {X 0,Y 333.667,Z 389.551,A -85,B 0,C 180,E1 -14436.14,E2 -14436.14} C_VEL
LIN {X 0,Y 333.596,Z 389.545,A -85,B 0,C 180,E1 -14439.199,E2 -14439.199} C_VEL
LIN {X 0,Y 333.621,Z 389.543,A -85,B 0,C 180,E1 -14442.499,E2 -14442.499} C_VEL
LIN {X 0,Y 333.678,Z 389.731,A -85,B 0,C 180,E1 -14447.022,E2 -14447.022} C_VEL
LIN {X 0,Y 337.792,Z 403.697,A -85,B 0,C 180,E1 -14450.028,E2 -14450.028} C_VEL
LIN {X 0,Y 341.569,Z 417.845,A -85,B 0,C 180,E1 -14452.873,E2 -14452.873} C_VEL
LIN {X 0,Y 344.391,Z 429.858,A -85,B 0,C 180,E1 -14455.153,E2 -14455.153} C_VEL
LIN {X 0,Y 343.736,Z 436.031,A -85,B 0,C 180,E1 -14456.141,E2 -14456.141} C_VEL
LIN {X 0,Y 342.997,Z 442.371,A -85,B 0,C 180,E1 -14457.149,E2 -14457.149} C_VEL
LIN {X 0,Y 349.16,Z 489.558,A -85,B 0,C 180,E1 -14458.775,E2 -14458.775} C_VEL
LIN {X 0,Y 351.409,Z 508.847,A -85,B 0,C 180,E1 -14459.395,E2 -14459.395} C_VEL
LIN {X 0,Y 348.692,Z 612.255,A -85,B 0,C 180,E1 -14461.524,E2 -14461.524} C_VEL
LIN {X 0,Y 347.726,Z 627.725,A -85,B 0,C 180,E1 -14462.054,E2 -14462.054} C_VEL
LIN {X 0,Y 346.188,Z 643.329,A -85,B 0,C 180,E1 -14462.821,E2 -14462.821} C_VEL
LIN {X 0,Y 344.292,Z 658.04,A -85,B 0,C 180,E1 -14463.787,E2 -14463.787} C_VEL
LIN {X 0,Y 342.661,Z 670.241,A -85,B 0,C 180,E1 -14464.813,E2 -14464.813} C_VEL
LIN {X 0,Y 340.781,Z 683.091,A -85,B 0,C 180,E1 -14466.126,E2 -14466.126} C_VEL
LIN {X 0,Y 338.927,Z 695.047,A -85,B 0,C 180,E1 -14467.603,E2 -14467.603} C_VEL
LIN {X 0,Y 337.248,Z 706.197,A -85,B 0,C 180,E1 -14469.251,E2 -14469.251} C_VEL
LIN {X 0,Y 335.736,Z 716.527,A -85,B 0,C 180,E1 -14471.067,E2 -14471.067} C_VEL
LIN {X 0,Y 334.354,Z 726.649,A -85,B 0,C 180,E1 -14473.201,E2 -14473.201} C_VEL
LIN {X 0,Y 333.53,Z 735.141,A -85,B 0,C 180,E1 -14475.353,E2 -14475.353} C_VEL
LIN {X 0,Y 332.892,Z 743.057,A -85,B 0,C 180,E1 -14477.812,E2 -14477.812} C_VEL
LIN {X 0,Y 332.781,Z 749.391,A -85,B 0,C 180,E1 -14480.273,E2 -14480.273} C_VEL
LIN {X 0,Y 332.941,Z 754.394,A -85,B 0,C 180,E1 -14482.799,E2 -14482.799} C_VEL
LIN {X 0,Y 333.232,Z 757.758,A -85,B 0,C 180,E1 -14485.16,E2 -14485.16} C_VEL
LIN {X 0,Y 333.306,Z 759.903,A -85,B 0,C 180,E1 -14487.583,E2 -14487.583} C_VEL
LIN {X 0,Y 333.572,Z 760.543,A -85,B 0,C 180,E1 -14488.792,E2 -14488.792} C_VEL
LIN {X 0,Y 333.707,Z 760.858,A -85,B 0,C 180,E1 -14490,E2 -14490} C_VEL
LIN {X 0,Y 333.557,Z 760.829,A -85,B 0,C 180,E1 -14491.207,E2 -14491.207} C_VEL
LIN {X 0,Y 333.167,Z 759.858,A -85,B 0,C 180,E1 -14493.628,E2 -14493.628} C_VEL
LIN {X 0,Y 333.078,Z 758.932,A -85,B 0,C 180,E1 -14494.841,E2 -14494.841} C_VEL
LIN {X 0,Y 332.786,Z 756.088,A -85,B 0,C 180,E1 -14497.279,E2 -14497.279} C_VEL
LIN {X 0,Y 332.619,Z 751.987,A -85,B 0,C 180,E1 -14499.731,E2 -14499.731} C_VEL
LIN {X 0,Y 332.791,Z 746.579,A -85,B 0,C 180,E1 -14502.191,E2 -14502.191} C_VEL
LIN {X 0,Y 333.468,Z 739.757,A -85,B 0,C 180,E1 -14504.649,E2 -14504.649} C_VEL
LIN {X 0,Y 334.573,Z 731.337,A -85,B 0,C 180,E1 -14507.102,E2 -14507.102} C_VEL
LIN {X 0,Y 336.198,Z 722.492,A -85,B 0,C 180,E1 -14509.222,E2 -14509.222} C_VEL
LIN {X 0,Y 338.124,Z 711.929,A -85,B 0,C 180,E1 -14511.329,E2 -14511.329} C_VEL
LIN {X 0,Y 340.251,Z 701.23,A -85,B 0,C 180,E1 -14513.106,E2 -14513.106} C_VEL
LIN {X 0,Y 342.555,Z 689.697,A -85,B 0,C 180,E1 -14514.709,E2 -14514.709} C_VEL
LIN {X 0,Y 345.21,Z 676.14,A -85,B 0,C 180,E1 -14516.246,E2 -14516.246} C_VEL
LIN {X 0,Y 347.731,Z 662.171,A -85,B 0,C 180,E1 -14517.52,E2 -14517.52} C_VEL
LIN {X 0,Y 350.13,Z 647.697,A -85,B 0,C 180,E1 -14518.552,E2 -14518.552} C_VEL
LIN {X 0,Y 352.154,Z 632.992,A -85,B 0,C 180,E1 -14519.352,E2 -14519.352} C_VEL
LIN {X 0,Y 353.663,Z 617.895,A -85,B 0,C 180,E1 -14519.951,E2 -14519.951} C_VEL
LIN {X 0,Y 354.534,Z 602.298,A -85,B 0,C 180,E1 -14520.363,E2 -14520.363} C_VEL
LIN {X 0,Y 357.403,Z 509.33,A -85,B 0,C 180,E1 -14522.269,E2 -14522.269} C_VEL
LIN {X 0,Y 354.305,Z 483.599,A -85,B 0,C 180,E1 -14523.242,E2 -14523.242} C_VEL
LIN {X 0,Y 349.898,Z 455.232,A -85,B 0,C 180,E1 -14524.47,E2 -14524.47} C_VEL
LIN {X 0,Y 347.163,Z 439.617,A -85,B 0,C 180,E1 -14525.235,E2 -14525.235} C_VEL
LIN {X 0,Y 347.568,Z 437.072,A -85,B 0,C 180,E1 -14525.654,E2 -14525.654} C_VEL
LIN {X 0,Y 346.586,Z 431.455,A -85,B 0,C 180,E1 -14526.777,E2 -14526.777} C_VEL
LIN {X 0,Y 342.794,Z 417.483,A -85,B 0,C 180,E1 -14529.836,E2 -14529.836} C_VEL
LIN {X 0,Y 338.694,Z 404.309,A -85,B 0,C 180,E1 -14532.993,E2 -14532.993} C_VEL
LIN {X 0,Y 334.602,Z 392.46,A -85,B 0,C 180,E1 -14536.122,E2 -14536.122} C_VEL
LIN {X 0,Y 333.636,Z 389.54,A -85,B 0,C 180,E1 -14536.992,E2 -14536.992} C_VEL
LIN {X 0,Y 333.606,Z 389.548,A -85,B 0,C 180,E1 -14541.209,E2 -14541.209} C_VEL
LIN {X 0,Y 333.663,Z 389.542,A -85,B 0,C 180,E1 -14543.86,E2 -14543.86} C_VEL
LIN {X 0,Y 333.634,Z 389.551,A -85,B 0,C 180,E1 -14547.413,E2 -14547.413} C_VEL
LIN {X 0,Y 333.64,Z 389.553,A -85,B 0,C 180,E1 -14551.022,E2 -14551.022} C_VEL
LIN {X 0,Y 333.649,Z 389.548,A -85,B 0,C 180,E1 -14555.085,E2 -14555.085} C_VEL
LIN {X 0,Y 333.626,Z 389.547,A -85,B 0,C 180,E1 -14559.016,E2 -14559.016} C_VEL
LIN {X 0,Y 333.693,Z 389.545,A -85,B 0,C 180,E1 -14561.584,E2 -14561.584} C_VEL
LIN {X 0,Y 333.749,Z 389.534,A -85,B 0,C 180,E1 -14565.609,E2 -14565.609} C_VEL
LIN {X 0,Y 333.802,Z 389.526,A -85,B 0,C 180,E1 -14569.077,E2 -14569.077} C_VEL
LIN {X 0,Y 333.941,Z 389.508,A -85,B 0,C 180,E1 -14572.746,E2 -14572.746} C_VEL
LIN {X 0,Y 333.769,Z 389.534,A -85,B 0,C 180,E1 -14575.169,E2 -14575.169} C_VEL
LIN {X 0,Y 334.056,Z 389.489,A -85,B 0,C 180,E1 -14577.589,E2 -14577.589} C_VEL
LIN {X 0,Y 334.067,Z 389.488,A -85,B 0,C 180,E1 -14581.206,E2 -14581.206} C_VEL
LIN {X 0,Y 333.794,Z 389.53,A -85,B 0,C 180,E1 -14583.622,E2 -14583.622} C_VEL
LIN {X 0,Y 333.949,Z 389.476,A -85,B 0,C 180,E1 -14586.709,E2 -14586.709} C_VEL
LIN {X 0,Y 333.808,Z 389.525,A -85,B 0,C 180,E1 -14589.697,E2 -14589.697} C_VEL
LIN {X 0,Y 333.782,Z 389.508,A -85,B 0,C 180,E1 -14593.392,E2 -14593.392} C_VEL
LIN {X 0,Y 333.747,Z 389.522,A -85,B 0,C 180,E1 -14595.888,E2 -14595.888} C_VEL
LIN {X 0,Y 333.674,Z 389.529,A -85,B 0,C 180,E1 -14599.695,E2 -14599.695} C_VEL
LIN {X 0,Y 333.632,Z 389.551,A -85,B 0,C 180,E1 -14603.593,E2 -14603.593} C_VEL
LIN {X 0,Y 333.619,Z 389.534,A -85,B 0,C 180,E1 -14606.257,E2 -14606.257} C_VEL
LIN {X 0,Y 333.641,Z 389.551,A -85,B 0,C 180,E1 -14608.979,E2 -14608.979} C_VEL
LIN {X 0,Y 333.635,Z 389.536,A -85,B 0,C 180,E1 -14612.588,E2 -14612.588} C_VEL
LIN {X 0,Y 333.666,Z 389.537,A -85,B 0,C 180,E1 -14616.141,E2 -14616.141} C_VEL
LIN {X 0,Y 333.613,Z 389.553,A -85,B 0,C 180,E1 -14619.198,E2 -14619.198} C_VEL
LIN {X 0,Y 333.623,Z 389.555,A -85,B 0,C 180,E1 -14622.5,E2 -14622.5} C_VEL
LIN {X 0,Y 333.601,Z 389.629,A -85,B 0,C 180,E1 -14624.596,E2 -14624.596} C_VEL
LIN {X 0,Y 334.603,Z 392.427,A -85,B 0,C 180,E1 -14624.823,E2 -14624.823} C_VEL
LIN {X 0,Y 336.446,Z 394.669,A -85,B 0,C 180,E1 -14625.154,E2 -14625.154} C_VEL
LIN {X 0,Y 338.595,Z 398.018,A -85,B 0,C 180,E1 -14625.554,E2 -14625.554} C_VEL
LIN {X 0,Y 348.567,Z 413.974,A -85,B 0,C 180,E1 -14627.32,E2 -14627.32} C_VEL
LIN {X 0,Y 357.325,Z 429.443,A -85,B 0,C 180,E1 -14628.792,E2 -14628.792} C_VEL
LIN {X 0,Y 359.407,Z 433.36,A -85,B 0,C 180,E1 -14629.133,E2 -14629.133} C_VEL
LIN {X 0,Y 357.654,Z 487.936,A -85,B 0,C 180,E1 -14630.253,E2 -14630.253} C_VEL
LIN {X 0,Y 356.95,Z 522.706,A -85,B 0,C 180,E1 -14631.039,E2 -14631.039} C_VEL
LIN {X 0,Y 356.281,Z 536.886,A -85,B 0,C 180,E1 -14631.541,E2 -14631.541} C_VEL
LIN {X 0,Y 355.41,Z 551.189,A -85,B 0,C 180,E1 -14632.277,E2 -14632.277} C_VEL
LIN {X 0,Y 354.201,Z 563.137,A -85,B 0,C 180,E1 -14633.049,E2 -14633.049} C_VEL
LIN {X 0,Y 352.575,Z 576.75,A -85,B 0,C 180,E1 -14634.16,E2 -14634.16} C_VEL
LIN {X 0,Y 350.762,Z 589.131,A -85,B 0,C 180,E1 -14635.402,E2 -14635.402} C_VEL
LIN {X 0,Y 348.677,Z 601.123,A -85,B 0,C 180,E1 -14636.858,E2 -14636.858} C_VEL
LIN {X 0,Y 346.417,Z 612.972,A -85,B 0,C 180,E1 -14638.617,E2 -14638.617} C_VEL
LIN {X 0,Y 344.332,Z 622.631,A -85,B 0,C 180,E1 -14640.335,E2 -14640.335} C_VEL
LIN {X 0,Y 342.008,Z 632.896,A -85,B 0,C 180,E1 -14642.549,E2 -14642.549} C_VEL
LIN {X 0,Y 340.13,Z 640.701,A -85,B 0,C 180,E1 -14644.613,E2 -14644.613} C_VEL
LIN {X 0,Y 338.448,Z 647.375,A -85,B 0,C 180,E1 -14646.764,E2 -14646.764} C_VEL
LIN {X 0,Y 336.945,Z 653.482,A -85,B 0,C 180,E1 -14649.233,E2 -14649.233} C_VEL
LIN {X 0,Y 335.715,Z 658.137,A -85,B 0,C 180,E1 -14651.7,E2 -14651.7} C_VEL
LIN {X 0,Y 334.814,Z 661.479,A -85,B 0,C 180,E1 -14654.165,E2 -14654.165} C_VEL
LIN {X 0,Y 334.213,Z 663.614,A -85,B 0,C 180,E1 -14656.626,E2 -14656.626} C_VEL
LIN {X 0,Y 333.976,Z 664.595,A -85,B 0,C 180,E1 -14659.084,E2 -14659.084} C_VEL
LIN {X 0,Y 333.893,Z 664.444,A -85,B 0,C 180,E1 -14661.608,E2 -14661.608} C_VEL
LIN {X 0,Y 333.915,Z 663.213,A -85,B 0,C 180,E1 -14663.96,E2 -14663.96} C_VEL
LIN {X 0,Y 334.137,Z 660.848,A -85,B 0,C 180,E1 -14666.383,E2 -14666.383} C_VEL
LIN {X 0,Y 334.639,Z 657.318,A -85,B 0,C 180,E1 -14668.797,E2 -14668.797} C_VEL
LIN {X 0,Y 335.38,Z 652.558,A -85,B 0,C 180,E1 -14671.201,E2 -14671.201} C_VEL
LIN {X 0,Y 336.44,Z 646.434,A -85,B 0,C 180,E1 -14673.593,E2 -14673.593} C_VEL
LIN {X 0,Y 337.698,Z 638.789,A -85,B 0,C 180,E1 -14675.973,E2 -14675.973} C_VEL
LIN {X 0,Y 339.114,Z 630.639,A -85,B 0,C 180,E1 -14678.042,E2 -14678.042} C_VEL
LIN {X 0,Y 340.804,Z 620.83,A -85,B 0,C 180,E1 -14680.095,E2 -14680.095} C_VEL
LIN {X 0,Y 342.38,Z 610.842,A -85,B 0,C 180,E1 -14681.845,E2 -14681.845} C_VEL
LIN {X 0,Y 344.01,Z 598.911,A -85,B 0,C 180,E1 -14683.588,E2 -14683.588} C_VEL
LIN {X 0,Y 345.565,Z 586.965,A -85,B 0,C 180,E1 -14685.029,E2 -14685.029} C_VEL
LIN {X 0,Y 347.113,Z 573.901,A -85,B 0,C 180,E1 -14686.316,E2 -14686.316} C_VEL
LIN {X 0,Y 348.561,Z 559.421,A -85,B 0,C 180,E1 -14687.453,E2 -14687.453} C_VEL
LIN {X 0,Y 349.661,Z 544.078,A -85,B 0,C 180,E1 -14688.38,E2 -14688.38} C_VEL
LIN {X 0,Y 350.348,Z 529.158,A -85,B 0,C 180,E1 -14689.038,E2 -14689.038} C_VEL
LIN {X 0,Y 350.611,Z 513.612,A -85,B 0,C 180,E1 -14689.492,E2 -14689.492} C_VEL
LIN {X 0,Y 352.333,Z 442.453,A -85,B 0,C 180,E1 -14690.956,E2 -14690.956} C_VEL
LIN {X 0,Y 352.019,Z 438.623,A -85,B 0,C 180,E1 -14691.07,E2 -14691.07} C_VEL
LIN {X 0,Y 350.984,Z 434.988,A -85,B 0,C 180,E1 -14691.242,E2 -14691.242} C_VEL
LIN {X 0,Y 348.528,Z 429.929,A -85,B 0,C 180,E1 -14691.574,E2 -14691.574} C_VEL
LIN {X 0,Y 341.203,Z 418.771,A -85,B 0,C 180,E1 -14692.504,E2 -14692.504} C_VEL
LIN {X 0,Y 339.4,Z 415.35,A -85,B 0,C 180,E1 -14692.756,E2 -14692.756} C_VEL
LIN {X 0,Y 329.726,Z 396.923,A -85,B 0,C 180,E1 -14694.169,E2 -14694.169} C_VEL
LIN {X 0,Y 326.853,Z 391.52,A -85,B 0,C 180,E1 -14694.606,E2 -14694.606} C_VEL
LIN {X 0,Y 326.623,Z 390.425,A -85,B 0,C 180,E1 -14694.683,E2 -14694.683} C_VEL
LIN {X 0,Y 326.589,Z 390.43,A -85,B 0,C 180,E1 -14698.257,E2 -14698.257} C_VEL
LIN {X 0,Y 326.571,Z 390.42,A -85,B 0,C 180,E1 -14701.097,E2 -14701.097} C_VEL
LIN {X 0,Y 326.606,Z 390.423,A -85,B 0,C 180,E1 -14704.019,E2 -14704.019} C_VEL
LIN {X 0,Y 326.621,Z 390.422,A -85,B 0,C 180,E1 -14707.236,E2 -14707.236} C_VEL
LIN {X 0,Y 326.533,Z 390.433,A -85,B 0,C 180,E1 -14711.122,E2 -14711.122} C_VEL
LIN {X 0,Y 326.517,Z 390.434,A -85,B 0,C 180,E1 -14714.74,E2 -14714.74} C_VEL
LIN {X 0,Y 326.558,Z 390.428,A -85,B 0,C 180,E1 -14718.151,E2 -14718.151} C_VEL
LIN {X 0,Y 326.564,Z 390.426,A -85,B 0,C 180,E1 -14721.383,E2 -14721.383} C_VEL
LIN {X 0,Y 326.615,Z 390.428,A -85,B 0,C 180,E1 -14724.851,E2 -14724.851} C_VEL
LIN {X 0,Y 326.598,Z 390.426,A -85,B 0,C 180,E1 -14727.454,E2 -14727.454} C_VEL
LIN {X 0,Y 326.571,Z 390.425,A -85,B 0,C 180,E1 -14730.332,E2 -14730.332} C_VEL
LIN {X 0,Y 326.6,Z 390.429,A -85,B 0,C 180,E1 -14733.134,E2 -14733.134} C_VEL
LIN {X 0,Y 326.626,Z 390.414,A -85,B 0,C 180,E1 -14735.869,E2 -14735.869} C_VEL
LIN {X 0,Y 326.61,Z 390.421,A -85,B 0,C 180,E1 -14739.861,E2 -14739.861} C_VEL
LIN {X 0,Y 326.702,Z 390.415,A -85,B 0,C 180,E1 -14743.76,E2 -14743.76} C_VEL
LIN {X 0,Y 326.75,Z 390.395,A -85,B 0,C 180,E1 -14746.314,E2 -14746.314} C_VEL
LIN {X 0,Y 326.775,Z 390.363,A -85,B 0,C 180,E1 -14750.092,E2 -14750.092} C_VEL
LIN {X 0,Y 326.932,Z 390.387,A -85,B 0,C 180,E1 -14753.829,E2 -14753.829} C_VEL
LIN {X 0,Y 327.033,Z 390.362,A -85,B 0,C 180,E1 -14758.768,E2 -14758.768} C_VEL
LIN {X 0,Y 327.003,Z 390.37,A -85,B 0,C 180,E1 -14762.463,E2 -14762.463} C_VEL
LIN {X 0,Y 326.928,Z 390.385,A -85,B 0,C 180,E1 -14766.17,E2 -14766.17} C_VEL
LIN {X 0,Y 326.775,Z 390.397,A -85,B 0,C 180,E1 -14769.907,E2 -14769.907} C_VEL
LIN {X 0,Y 326.726,Z 390.404,A -85,B 0,C 180,E1 -14773.686,E2 -14773.686} C_VEL
LIN {X 0,Y 326.615,Z 390.425,A -85,B 0,C 180,E1 -14777.532,E2 -14777.532} C_VEL
LIN {X 0,Y 326.6,Z 390.43,A -85,B 0,C 180,E1 -14781.458,E2 -14781.458} C_VEL
LIN {X 0,Y 326.593,Z 390.428,A -85,B 0,C 180,E1 -14785.492,E2 -14785.492} C_VEL
LIN {X 0,Y 326.584,Z 390.429,A -85,B 0,C 180,E1 -14788.257,E2 -14788.257} C_VEL
LIN {X 0,Y 326.568,Z 390.433,A -85,B 0,C 180,E1 -14791.097,E2 -14791.097} C_VEL
LIN {X 0,Y 326.601,Z 390.412,A -85,B 0,C 180,E1 -14794.02,E2 -14794.02} C_VEL
LIN {X 0,Y 326.616,Z 390.423,A -85,B 0,C 180,E1 -14797.237,E2 -14797.237} C_VEL
LIN {X 0,Y 326.538,Z 390.435,A -85,B 0,C 180,E1 -14801.124,E2 -14801.124} C_VEL
LIN {X 0,Y 326.554,Z 390.431,A -85,B 0,C 180,E1 -14803.527,E2 -14803.527} C_VEL
LIN {X 0,Y 326.59,Z 390.55,A -85,B 0,C 180,E1 -14806.374,E2 -14806.374} C_VEL
LIN {X 0,Y 330.695,Z 404.334,A -85,B 0,C 180,E1 -14809.443,E2 -14809.443} C_VEL
LIN {X 0,Y 334.64,Z 418.992,A -85,B 0,C 180,E1 -14812.48,E2 -14812.48} C_VEL
LIN {X 0,Y 337.391,Z 430.561,A -85,B 0,C 180,E1 -14814.737,E2 -14814.737} C_VEL
LIN {X 0,Y 337.668,Z 432.452,A -85,B 0,C 180,E1 -14815.085,E2 -14815.085} C_VEL
LIN {X 0,Y 336.432,Z 441.273,A -85,B 0,C 180,E1 -14816.508,E2 -14816.508} C_VEL
LIN {X 0,Y 340.731,Z 473.748,A -85,B 0,C 180,E1 -14817.68,E2 -14817.68} C_VEL
LIN {X 0,Y 345.049,Z 509.212,A -85,B 0,C 180,E1 -14818.878,E2 -14818.878} C_VEL
LIN {X 0,Y 342.25,Z 611.511,A -85,B 0,C 180,E1 -14821.021,E2 -14821.021} C_VEL
LIN {X 0,Y 341.176,Z 627.685,A -85,B 0,C 180,E1 -14821.594,E2 -14821.594} C_VEL
LIN {X 0,Y 339.651,Z 642.444,A -85,B 0,C 180,E1 -14822.337,E2 -14822.337} C_VEL
LIN {X 0,Y 337.764,Z 656.973,A -85,B 0,C 180,E1 -14823.309,E2 -14823.309} C_VEL
LIN {X 0,Y 335.92,Z 670.133,A -85,B 0,C 180,E1 -14824.437,E2 -14824.437} C_VEL
LIN {X 0,Y 333.802,Z 684.142,A -85,B 0,C 180,E1 -14825.925,E2 -14825.925} C_VEL
LIN {X 0,Y 331.725,Z 696.843,A -85,B 0,C 180,E1 -14827.583,E2 -14827.583} C_VEL
LIN {X 0,Y 329.915,Z 708.318,A -85,B 0,C 180,E1 -14829.397,E2 -14829.397} C_VEL
LIN {X 0,Y 328.212,Z 719.774,A -85,B 0,C 180,E1 -14831.588,E2 -14831.588} C_VEL
LIN {X 0,Y 326.977,Z 729.203,A -85,B 0,C 180,E1 -14833.774,E2 -14833.774} C_VEL
LIN {X 0,Y 326.124,Z 738.078,A -85,B 0,C 180,E1 -14836.287,E2 -14836.287} C_VEL
LIN {X 0,Y 325.707,Z 745.223,A -85,B 0,C 180,E1 -14838.802,E2 -14838.802} C_VEL
LIN {X 0,Y 325.766,Z 750.864,A -85,B 0,C 180,E1 -14841.314,E2 -14841.314} C_VEL
LIN {X 0,Y 325.964,Z 755.061,A -85,B 0,C 180,E1 -14843.811,E2 -14843.811} C_VEL
LIN {X 0,Y 326.174,Z 756.662,A -85,B 0,C 180,E1 -14845.055,E2 -14845.055} C_VEL
LIN {X 0,Y 326.271,Z 758.845,A -85,B 0,C 180,E1 -14847.53,E2 -14847.53} C_VEL
LIN {X 0,Y 326.542,Z 759.502,A -85,B 0,C 180,E1 -14848.766,E2 -14848.766} C_VEL
LIN {X 0,Y 326.698,Z 759.836,A -85,B 0,C 180,E1 -14850,E2 -14850} C_VEL
LIN {X 0,Y 326.525,Z 759.82,A -85,B 0,C 180,E1 -14851.233,E2 -14851.233} C_VEL
LIN {X 0,Y 326.119,Z 758.876,A -85,B 0,C 180,E1 -14853.706,E2 -14853.706} C_VEL
LIN {X 0,Y 326.014,Z 757.952,A -85,B 0,C 180,E1 -14854.946,E2 -14854.946} C_VEL
LIN {X 0,Y 325.688,Z 755.126,A -85,B 0,C 180,E1 -14857.438,E2 -14857.438} C_VEL
LIN {X 0,Y 325.544,Z 751.058,A -85,B 0,C 180,E1 -14859.945,E2 -14859.945} C_VEL
LIN {X 0,Y 325.733,Z 745.683,A -85,B 0,C 180,E1 -14862.459,E2 -14862.459} C_VEL
LIN {X 0,Y 326.481,Z 738.901,A -85,B 0,C 180,E1 -14864.969,E2 -14864.969} C_VEL
LIN {X 0,Y 327.692,Z 730.526,A -85,B 0,C 180,E1 -14867.472,E2 -14867.472} C_VEL
LIN {X 0,Y 329.402,Z 721.733,A -85,B 0,C 180,E1 -14869.635,E2 -14869.635} C_VEL
LIN {X 0,Y 331.097,Z 712.893,A -85,B 0,C 180,E1 -14871.478,E2 -14871.478} C_VEL
LIN {X 0,Y 333.645,Z 700.619,A -85,B 0,C 180,E1 -14873.591,E2 -14873.591} C_VEL
LIN {X 0,Y 336.096,Z 689.169,A -85,B 0,C 180,E1 -14875.216,E2 -14875.216} C_VEL
LIN {X 0,Y 338.817,Z 675.775,A -85,B 0,C 180,E1 -14876.776,E2 -14876.776} C_VEL
LIN {X 0,Y 341.464,Z 661.745,A -85,B 0,C 180,E1 -14878.086,E2 -14878.086} C_VEL
LIN {X 0,Y 343.904,Z 647.651,A -85,B 0,C 180,E1 -14879.118,E2 -14879.118} C_VEL
LIN {X 0,Y 345.999,Z 633.221,A -85,B 0,C 180,E1 -14879.927,E2 -14879.927} C_VEL
LIN {X 0,Y 347.643,Z 617.665,A -85,B 0,C 180,E1 -14880.567,E2 -14880.567} C_VEL
LIN {X 0,Y 348.571,Z 602.549,A -85,B 0,C 180,E1 -14880.981,E2 -14880.981} C_VEL
LIN {X 0,Y 351.557,Z 510.403,A -85,B 0,C 180,E1 -14882.9,E2 -14882.9} C_VEL
LIN {X 0,Y 348.547,Z 484.849,A -85,B 0,C 180,E1 -14883.888,E2 -14883.888} C_VEL
LIN {X 0,Y 344.217,Z 456.634,A -85,B 0,C 180,E1 -14885.145,E2 -14885.145} C_VEL
LIN {X 0,Y 340.976,Z 438.437,A -85,B 0,C 180,E1 -14886.07,E2 -14886.07} C_VEL
LIN {X 0,Y 338.885,Z 429.425,A -85,B 0,C 180,E1 -14887.995,E2 -14887.995} C_VEL
LIN {X 0,Y 335.253,Z 416.329,A -85,B 0,C 180,E1 -14891.003,E2 -14891.003} C_VEL
LIN {X 0,Y 331.192,Z 403.628,A -85,B 0,C 180,E1 -14894.206,E2 -14894.206} C_VEL
LIN {X 0,Y 327.305,Z 392.733,A -85,B 0,C 180,E1 -14897.239,E2 -14897.239} C_VEL
LIN {X 0,Y 326.561,Z 390.43,A -85,B 0,C 180,E1 -14897.959,E2 -14897.959} C_VEL
LIN {X 0,Y 326.557,Z 390.426,A -85,B 0,C 180,E1 -14901.382,E2 -14901.382} C_VEL
LIN {X 0,Y 326.608,Z 390.428,A -85,B 0,C 180,E1 -14904.851,E2 -14904.851} C_VEL
LIN {X 0,Y 326.598,Z 390.428,A -85,B 0,C 180,E1 -14907.455,E2 -14907.455} C_VEL
LIN {X 0,Y 326.605,Z 390.426,A -85,B 0,C 180,E1 -14910.336,E2 -14910.336} C_VEL
LIN {X 0,Y 326.588,Z 390.432,A -85,B 0,C 180,E1 -14914.508,E2 -14914.508} C_VEL
LIN {X 0,Y 326.59,Z 390.426,A -85,B 0,C 180,E1 -14918.542,E2 -14918.542} C_VEL
LIN {X 0,Y 326.609,Z 390.422,A -85,B 0,C 180,E1 -14922.467,E2 -14922.467} C_VEL
LIN {X 0,Y 326.721,Z 390.407,A -85,B 0,C 180,E1 -14926.313,E2 -14926.313} C_VEL
LIN {X 0,Y 326.77,Z 390.399,A -85,B 0,C 180,E1 -14930.093,E2 -14930.093} C_VEL
LIN {X 0,Y 326.925,Z 390.377,A -85,B 0,C 180,E1 -14933.83,E2 -14933.83} C_VEL
LIN {X 0,Y 327,Z 390.367,A -85,B 0,C 180,E1 -14937.537,E2 -14937.537} C_VEL
LIN {X 0,Y 327.035,Z 390.364,A -85,B 0,C 180,E1 -14941.232,E2 -14941.232} C_VEL
LIN {X 0,Y 326.743,Z 390.408,A -85,B 0,C 180,E1 -14943.7,E2 -14943.7} C_VEL
LIN {X 0,Y 326.907,Z 390.353,A -85,B 0,C 180,E1 -14946.702,E2 -14946.702} C_VEL
LIN {X 0,Y 326.771,Z 390.402,A -85,B 0,C 180,E1 -14949.908,E2 -14949.908} C_VEL
LIN {X 0,Y 326.746,Z 390.381,A -85,B 0,C 180,E1 -14953.686,E2 -14953.686} C_VEL
LIN {X 0,Y 326.654,Z 390.42,A -85,B 0,C 180,E1 -14957.531,E2 -14957.531} C_VEL
LIN {X 0,Y 326.617,Z 390.402,A -85,B 0,C 180,E1 -14960.138,E2 -14960.138} C_VEL
LIN {X 0,Y 326.6,Z 390.428,A -85,B 0,C 180,E1 -14964.133,E2 -14964.133} C_VEL
LIN {X 0,Y 326.587,Z 390.421,A -85,B 0,C 180,E1 -14968.258,E2 -14968.258} C_VEL
LIN {X 0,Y 326.562,Z 390.42,A -85,B 0,C 180,E1 -14971.099,E2 -14971.099} C_VEL
LIN {X 0,Y 326.598,Z 390.431,A -85,B 0,C 180,E1 -14974.021,E2 -14974.021} C_VEL
LIN {X 0,Y 326.615,Z 390.415,A -85,B 0,C 180,E1 -14977.238,E2 -14977.238} C_VEL
LIN {X 0,Y 326.537,Z 390.425,A -85,B 0,C 180,E1 -14981.126,E2 -14981.126} C_VEL
LIN {X 0,Y 326.531,Z 390.426,A -85,B 0,C 180,E1 -14983.531,E2 -14983.531} C_VEL
LIN {X 0,Y 327.563,Z 393.317,A -85,B 0,C 180,E1 -14983.78,E2 -14983.78} C_VEL
LIN {X 0,Y 329.526,Z 395.732,A -85,B 0,C 180,E1 -14984.153,E2 -14984.153} C_VEL
LIN {X 0,Y 331.677,Z 399.046,A -85,B 0,C 180,E1 -14984.573,E2 -14984.573} C_VEL
LIN {X 0,Y 340.305,Z 412.465,A -85,B 0,C 180,E1 -14986.182,E2 -14986.182} C_VEL
LIN {X 0,Y 350.162,Z 429.318,A -85,B 0,C 180,E1 -14987.915,E2 -14987.915} C_VEL
LIN {X 0,Y 353.681,Z 436.272,A -85,B 0,C 180,E1 -14988.524,E2 -14988.524} C_VEL
LIN {X 0,Y 351.331,Z 508.524,A -85,B 0,C 180,E1 -14990.034,E2 -14990.034} C_VEL
LIN {X 0,Y 350.93,Z 527.268,A -85,B 0,C 180,E1 -14990.519,E2 -14990.519} C_VEL
LIN {X 0,Y 350.192,Z 541.652,A -85,B 0,C 180,E1 -14991.092,E2 -14991.092} C_VEL
LIN {X 0,Y 349.21,Z 555.159,A -85,B 0,C 180,E1 -14991.839,E2 -14991.839} C_VEL
LIN {X 0,Y 347.891,Z 567.366,A -85,B 0,C 180,E1 -14992.697,E2 -14992.697} C_VEL
LIN {X 0,Y 345.999,Z 581.305,A -85,B 0,C 180,E1 -14993.912,E2 -14993.912} C_VEL
LIN {X 0,Y 343.936,Z 593.96,A -85,B 0,C 180,E1 -14995.279,E2 -14995.279} C_VEL
LIN {X 0,Y 341.753,Z 605.577,A -85,B 0,C 180,E1 -14996.804,E2 -14996.804} C_VEL
LIN {X 0,Y 339.463,Z 616.853,A -85,B 0,C 180,E1 -14998.599,E2 -14998.599} C_VEL
LIN {X 0,Y 337.344,Z 626.061,A -85,B 0,C 180,E1 -15000.345,E2 -15000.345} C_VEL
LIN {X 0,Y 335.044,Z 635.544,A -85,B 0,C 180,E1 -15002.519,E2 -15002.519} C_VEL
LIN {X 0,Y 333.337,Z 642.359,A -85,B 0,C 180,E1 -15004.393,E2 -15004.393} C_VEL
LIN {X 0,Y 331.366,Z 649.762,A -85,B 0,C 180,E1 -15006.899,E2 -15006.899} C_VEL
LIN {X 0,Y 330.208,Z 654.228,A -85,B 0,C 180,E1 -15008.789,E2 -15008.789} C_VEL
LIN {X 0,Y 328.898,Z 658.952,A -85,B 0,C 180,E1 -15011.306,E2 -15011.306} C_VEL
LIN {X 0,Y 327.915,Z 662.361,A -85,B 0,C 180,E1 -15013.823,E2 -15013.823} C_VEL
LIN {X 0,Y 327.257,Z 664.56,A -85,B 0,C 180,E1 -15016.337,E2 -15016.337} C_VEL
LIN {X 0,Y 326.962,Z 665.606,A -85,B 0,C 180,E1 -15018.846,E2 -15018.846} C_VEL
LIN {X 0,Y 326.858,Z 665.473,A -85,B 0,C 180,E1 -15021.527,E2 -15021.527} C_VEL
LIN {X 0,Y 326.896,Z 664.309,A -85,B 0,C 180,E1 -15023.83,E2 -15023.83} C_VEL
LIN {X 0,Y 327.1,Z 662.008,A -85,B 0,C 180,E1 -15026.305,E2 -15026.305} C_VEL
LIN {X 0,Y 327.619,Z 658.542,A -85,B 0,C 180,E1 -15028.771,E2 -15028.771} C_VEL
LIN {X 0,Y 328.368,Z 653.852,A -85,B 0,C 180,E1 -15031.227,E2 -15031.227} C_VEL
LIN {X 0,Y 329.464,Z 647.8,A -85,B 0,C 180,E1 -15033.67,E2 -15033.67} C_VEL
LIN {X 0,Y 330.778,Z 640.232,A -85,B 0,C 180,E1 -15036.099,E2 -15036.099} C_VEL
LIN {X 0,Y 332.206,Z 632.179,A -85,B 0,C 180,E1 -15038.21,E2 -15038.21} C_VEL
LIN {X 0,Y 333.95,Z 622.474,A -85,B 0,C 180,E1 -15040.305,E2 -15040.305} C_VEL
LIN {X 0,Y 335.585,Z 612.578,A -85,B 0,C 180,E1 -15042.089,E2 -15042.089} C_VEL
LIN {X 0,Y 337.265,Z 600.808,A -85,B 0,C 180,E1 -15043.865,E2 -15043.865} C_VEL
LIN {X 0,Y 339.036,Z 587.721,A -85,B 0,C 180,E1 -15045.479,E2 -15045.479} C_VEL
LIN {X 0,Y 340.668,Z 574.603,A -85,B 0,C 180,E1 -15046.787,E2 -15046.787} C_VEL
LIN {X 0,Y 341.926,Z 562.02,A -85,B 0,C 180,E1 -15047.803,E2 -15047.803} C_VEL
LIN {X 0,Y 343.106,Z 547.225,A -85,B 0,C 180,E1 -15048.744,E2 -15048.744} C_VEL
LIN {X 0,Y 343.876,Z 532.028,A -85,B 0,C 180,E1 -15049.459,E2 -15049.459} C_VEL
LIN {X 0,Y 344.256,Z 516.709,A -85,B 0,C 180,E1 -15049.94,E2 -15049.94} C_VEL
LIN {X 0,Y 345.909,Z 447,A -85,B 0,C 180,E1 -15051.412,E2 -15051.412} C_VEL
LIN {X 0,Y 346.356,Z 430.017,A -85,B 0,C 180,E1 -15051.766,E2 -15051.766} C_VEL
LIN {X 0,Y 339.4,Z 415.35,A -85,B 0,C 180,E1 -15052.756,E2 -15052.756} C_VEL
LIN {X 0,Y 336.572,Z 410.724,A -85,B 0,C 180,E1 -15053.141,E2 -15053.141} C_VEL
LIN {X 0,Y 330.474,Z 404.372,A -85,B 0,C 180,E1 -15053.906,E2 -15053.906} C_VEL
LIN {X 0,Y 322.82,Z 397.061,A -85,B 0,C 180,E1 -15054.899,E2 -15054.899} C_VEL
LIN {X 0,Y 320.619,Z 394.243,A -85,B 0,C 180,E1 -15055.213,E2 -15055.213} C_VEL
LIN {X 0,Y 319.567,Z 391.306,A -85,B 0,C 180,E1 -15055.417,E2 -15055.417} C_VEL
LIN {X 0,Y 319.522,Z 391.298,A -85,B 0,C 180,E1 -15058.94,E2 -15058.94} C_VEL
LIN {X 0,Y 319.522,Z 391.311,A -85,B 0,C 180,E1 -15061.862,E2 -15061.862} C_VEL
LIN {X 0,Y 319.578,Z 391.302,A -85,B 0,C 180,E1 -15065.542,E2 -15065.542} C_VEL
LIN {X 0,Y 319.528,Z 391.301,A -85,B 0,C 180,E1 -15069.661,E2 -15069.661} C_VEL
LIN {X 0,Y 319.485,Z 391.307,A -85,B 0,C 180,E1 -15073.453,E2 -15073.453} C_VEL
LIN {X 0,Y 319.546,Z 391.301,A -85,B 0,C 180,E1 -15077.015,E2 -15077.015} C_VEL
LIN {X 0,Y 319.528,Z 391.308,A -85,B 0,C 180,E1 -15080.368,E2 -15080.368} C_VEL
LIN {X 0,Y 319.575,Z 391.303,A -85,B 0,C 180,E1 -15084.457,E2 -15084.457} C_VEL
LIN {X 0,Y 319.514,Z 391.31,A -85,B 0,C 180,E1 -15088.136,E2 -15088.136} C_VEL
LIN {X 0,Y 319.538,Z 391.302,A -85,B 0,C 180,E1 -15091.613,E2 -15091.613} C_VEL
LIN {X 0,Y 319.568,Z 391.296,A -85,B 0,C 180,E1 -15095.301,E2 -15095.301} C_VEL
LIN {X 0,Y 319.56,Z 391.304,A -85,B 0,C 180,E1 -15098.045,E2 -15098.045} C_VEL
LIN {X 0,Y 319.608,Z 391.293,A -85,B 0,C 180,E1 -15102.07,E2 -15102.07} C_VEL
LIN {X 0,Y 319.725,Z 391.271,A -85,B 0,C 180,E1 -15106.007,E2 -15106.007} C_VEL
LIN {X 0,Y 319.728,Z 391.238,A -85,B 0,C 180,E1 -15109.872,E2 -15109.872} C_VEL
LIN {X 0,Y 319.889,Z 391.262,A -85,B 0,C 180,E1 -15113.693,E2 -15113.693} C_VEL
LIN {X 0,Y 320,Z 391.238,A -85,B 0,C 180,E1 -15118.741,E2 -15118.741} C_VEL
LIN {X 0,Y 319.95,Z 391.248,A -85,B 0,C 180,E1 -15122.518,E2 -15122.518} C_VEL
LIN {X 0,Y 319.886,Z 391.261,A -85,B 0,C 180,E1 -15126.306,E2 -15126.306} C_VEL
LIN {X 0,Y 319.727,Z 391.276,A -85,B 0,C 180,E1 -15130.128,E2 -15130.128} C_VEL
LIN {X 0,Y 319.694,Z 391.278,A -85,B 0,C 180,E1 -15133.994,E2 -15133.994} C_VEL
LIN {X 0,Y 319.568,Z 391.298,A -85,B 0,C 180,E1 -15137.932,E2 -15137.932} C_VEL
LIN {X 0,Y 319.556,Z 391.301,A -85,B 0,C 180,E1 -15141.955,E2 -15141.955} C_VEL
LIN {X 0,Y 319.543,Z 391.301,A -85,B 0,C 180,E1 -15146.096,E2 -15146.096} C_VEL
LIN {X 0,Y 319.519,Z 391.308,A -85,B 0,C 180,E1 -15148.94,E2 -15148.94} C_VEL
LIN {X 0,Y 319.519,Z 391.308,A -85,B 0,C 180,E1 -15151.863,E2 -15151.863} C_VEL
LIN {X 0,Y 319.572,Z 391.302,A -85,B 0,C 180,E1 -15155.542,E2 -15155.542} C_VEL
LIN {X 0,Y 319.524,Z 391.302,A -85,B 0,C 180,E1 -15159.662,E2 -15159.662} C_VEL
LIN {X 0,Y 319.514,Z 391.306,A -85,B 0,C 180,E1 -15163.46,E2 -15163.46} C_VEL
LIN {X 0,Y 319.523,Z 391.39,A -85,B 0,C 180,E1 -15165.707,E2 -15165.707} C_VEL
LIN {X 0,Y 323.627,Z 404.836,A -85,B 0,C 180,E1 -15168.812,E2 -15168.812} C_VEL
LIN {X 0,Y 327.726,Z 420.105,A -85,B 0,C 180,E1 -15172.067,E2 -15172.067} C_VEL
LIN {X 0,Y 330.796,Z 433.493,A -85,B 0,C 180,E1 -15174.73,E2 -15174.73} C_VEL
LIN {X 0,Y 329.952,Z 440.576,A -85,B 0,C 180,E1 -15175.865,E2 -15175.865} C_VEL
LIN {X 0,Y 334.347,Z 473.353,A -85,B 0,C 180,E1 -15177.086,E2 -15177.086} C_VEL
LIN {X 0,Y 338.735,Z 510.906,A -85,B 0,C 180,E1 -15178.375,E2 -15178.375} C_VEL
LIN {X 0,Y 335.85,Z 610.713,A -85,B 0,C 180,E1 -15180.501,E2 -15180.501} C_VEL
LIN {X 0,Y 334.716,Z 626.8,A -85,B 0,C 180,E1 -15181.081,E2 -15181.081} C_VEL
LIN {X 0,Y 333.177,Z 641.534,A -85,B 0,C 180,E1 -15181.838,E2 -15181.838} C_VEL
LIN {X 0,Y 331.194,Z 656.124,A -85,B 0,C 180,E1 -15182.83,E2 -15182.83} C_VEL
LIN {X 0,Y 329.176,Z 670.077,A -85,B 0,C 180,E1 -15184.056,E2 -15184.056} C_VEL
LIN {X 0,Y 327.023,Z 683.807,A -85,B 0,C 180,E1 -15185.563,E2 -15185.563} C_VEL
LIN {X 0,Y 324.894,Z 696.4,A -85,B 0,C 180,E1 -15187.253,E2 -15187.253} C_VEL
LIN {X 0,Y 323.076,Z 707.396,A -85,B 0,C 180,E1 -15189.032,E2 -15189.032} C_VEL
LIN {X 0,Y 321.353,Z 718.43,A -85,B 0,C 180,E1 -15191.181,E2 -15191.181} C_VEL
LIN {X 0,Y 320.04,Z 727.904,A -85,B 0,C 180,E1 -15193.413,E2 -15193.413} C_VEL
LIN {X 0,Y 319.133,Z 736.846,A -85,B 0,C 180,E1 -15195.981,E2 -15195.981} C_VEL
LIN {X 0,Y 318.647,Z 744.032,A -85,B 0,C 180,E1 -15198.55,E2 -15198.55} C_VEL
LIN {X 0,Y 318.694,Z 749.709,A -85,B 0,C 180,E1 -15201.12,E2 -15201.12} C_VEL
LIN {X 0,Y 318.896,Z 753.941,A -85,B 0,C 180,E1 -15203.673,E2 -15203.673} C_VEL
LIN {X 0,Y 319.101,Z 755.56,A -85,B 0,C 180,E1 -15204.945,E2 -15204.945} C_VEL
LIN {X 0,Y 319.235,Z 757.786,A -85,B 0,C 180,E1 -15207.476,E2 -15207.476} C_VEL
LIN {X 0,Y 319.512,Z 758.461,A -85,B 0,C 180,E1 -15208.739,E2 -15208.739} C_VEL
LIN {X 0,Y 319.686,Z 758.814,A -85,B 0,C 180,E1 -15210,E2 -15210} C_VEL
LIN {X 0,Y 319.492,Z 758.811,A -85,B 0,C 180,E1 -15211.26,E2 -15211.26} C_VEL
LIN {X 0,Y 319.071,Z 757.893,A -85,B 0,C 180,E1 -15213.788,E2 -15213.788} C_VEL
LIN {X 0,Y 318.759,Z 755.719,A -85,B 0,C 180,E1 -15216.329,E2 -15216.329} C_VEL
LIN {X 0,Y 318.49,Z 752.304,A -85,B 0,C 180,E1 -15218.885,E2 -15218.885} C_VEL
LIN {X 0,Y 318.507,Z 747.624,A -85,B 0,C 180,E1 -15221.454,E2 -15221.454} C_VEL
LIN {X 0,Y 319.02,Z 741.599,A -85,B 0,C 180,E1 -15224.023,E2 -15224.023} C_VEL
LIN {X 0,Y 320.06,Z 734.092,A -85,B 0,C 180,E1 -15226.585,E2 -15226.585} C_VEL
LIN {X 0,Y 321.529,Z 726.182,A -85,B 0,C 180,E1 -15228.808,E2 -15228.808} C_VEL
LIN {X 0,Y 323.517,Z 716.42,A -85,B 0,C 180,E1 -15231.079,E2 -15231.079} C_VEL
LIN {X 0,Y 325.84,Z 705.495,A -85,B 0,C 180,E1 -15233.179,E2 -15233.179} C_VEL
LIN {X 0,Y 328.404,Z 694.03,A -85,B 0,C 180,E1 -15235.001,E2 -15235.001} C_VEL
LIN {X 0,Y 331.322,Z 680.967,A -85,B 0,C 180,E1 -15236.695,E2 -15236.695} C_VEL
LIN {X 0,Y 333.993,Z 667.814,A -85,B 0,C 180,E1 -15238.086,E2 -15238.086} C_VEL
LIN {X 0,Y 336.517,Z 654.418,A -85,B 0,C 180,E1 -15239.219,E2 -15239.219} C_VEL
LIN {X 0,Y 338.953,Z 639.762,A -85,B 0,C 180,E1 -15240.185,E2 -15240.185} C_VEL
LIN {X 0,Y 341.058,Z 623.764,A -85,B 0,C 180,E1 -15240.964,E2 -15240.964} C_VEL
LIN {X 0,Y 342.294,Z 608.646,A -85,B 0,C 180,E1 -15241.484,E2 -15241.484} C_VEL
LIN {X 0,Y 343.778,Z 569.107,A -85,B 0,C 180,E1 -15242.34,E2 -15242.34} C_VEL
LIN {X 0,Y 345.698,Z 511.002,A -85,B 0,C 180,E1 -15243.573,E2 -15243.573} C_VEL
LIN {X 0,Y 343.02,Z 487.628,A -85,B 0,C 180,E1 -15244.496,E2 -15244.496} C_VEL
LIN {X 0,Y 339.241,Z 462.003,A -85,B 0,C 180,E1 -15245.65,E2 -15245.65} C_VEL
LIN {X 0,Y 335.61,Z 441.616,A -85,B 0,C 180,E1 -15246.688,E2 -15246.688} C_VEL
LIN {X 0,Y 333.692,Z 437.094,A -85,B 0,C 180,E1 -15247.104,E2 -15247.104} C_VEL
LIN {X 0,Y 330.36,Z 424.269,A -85,B 0,C 180,E1 -15250.017,E2 -15250.017} C_VEL
LIN {X 0,Y 326.744,Z 412.212,A -85,B 0,C 180,E1 -15253.004,E2 -15253.004} C_VEL
LIN {X 0,Y 322.774,Z 400.536,A -85,B 0,C 180,E1 -15256.192,E2 -15256.192} C_VEL
LIN {X 0,Y 319.499,Z 391.306,A -85,B 0,C 180,E1 -15258.969,E2 -15258.969} C_VEL
LIN {X 0,Y 319.531,Z 391.309,A -85,B 0,C 180,E1 -15262.352,E2 -15262.352} C_VEL
LIN {X 0,Y 319.549,Z 391.307,A -85,B 0,C 180,E1 -15265.122,E2 -15265.122} C_VEL
LIN {X 0,Y 319.514,Z 391.314,A -85,B 0,C 180,E1 -15268.137,E2 -15268.137} C_VEL
LIN {X 0,Y 319.558,Z 391.307,A -85,B 0,C 180,E1 -15271.604,E2 -15271.604} C_VEL
LIN {X 0,Y 319.513,Z 391.307,A -85,B 0,C 180,E1 -15275.297,E2 -15275.297} C_VEL
LIN {X 0,Y 319.549,Z 391.308,A -85,B 0,C 180,E1 -15278.045,E2 -15278.045} C_VEL
LIN {X 0,Y 319.562,Z 391.301,A -85,B 0,C 180,E1 -15282.068,E2 -15282.068} C_VEL
LIN {X 0,Y 319.689,Z 391.283,A -85,B 0,C 180,E1 -15286.006,E2 -15286.006} C_VEL
LIN {X 0,Y 319.722,Z 391.276,A -85,B 0,C 180,E1 -15289.872,E2 -15289.872} C_VEL
LIN {X 0,Y 319.883,Z 391.254,A -85,B 0,C 180,E1 -15293.693,E2 -15293.693} C_VEL
LIN {X 0,Y 319.946,Z 391.246,A -85,B 0,C 180,E1 -15297.482,E2 -15297.482} C_VEL
LIN {X 0,Y 320.002,Z 391.24,A -85,B 0,C 180,E1 -15301.259,E2 -15301.259} C_VEL
LIN {X 0,Y 319.71,Z 391.271,A -85,B 0,C 180,E1 -15305.045,E2 -15305.045} C_VEL
LIN {X 0,Y 319.847,Z 391.232,A -85,B 0,C 180,E1 -15307.576,E2 -15307.576} C_VEL
LIN {X 0,Y 319.702,Z 391.284,A -85,B 0,C 180,E1 -15311.411,E2 -15311.411} C_VEL
LIN {X 0,Y 319.702,Z 391.255,A -85,B 0,C 180,E1 -15314.711,E2 -15314.711} C_VEL
LIN {X 0,Y 319.63,Z 391.285,A -85,B 0,C 180,E1 -15319.013,E2 -15319.013} C_VEL
LIN {X 0,Y 319.531,Z 391.307,A -85,B 0,C 180,E1 -15323.323,E2 -15323.323} C_VEL
LIN {X 0,Y 319.541,Z 391.288,A -85,B 0,C 180,E1 -15326.097,E2 -15326.097} C_VEL
LIN {X 0,Y 319.532,Z 391.308,A -85,B 0,C 180,E1 -15328.94,E2 -15328.94} C_VEL
LIN {X 0,Y 319.514,Z 391.293,A -85,B 0,C 180,E1 -15331.864,E2 -15331.864} C_VEL
LIN {X 0,Y 319.571,Z 391.298,A -85,B 0,C 180,E1 -15335.544,E2 -15335.544} C_VEL
LIN {X 0,Y 319.522,Z 391.303,A -85,B 0,C 180,E1 -15339.663,E2 -15339.663} C_VEL
LIN {X 0,Y 319.523,Z 391.408,A -85,B 0,C 180,E1 -15342.422,E2 -15342.422} C_VEL
LIN {X 0,Y 320.55,Z 394.173,A -85,B 0,C 180,E1 -15342.677,E2 -15342.677} C_VEL
LIN {X 0,Y 322.6,Z 396.753,A -85,B 0,C 180,E1 -15343.09,E2 -15343.09} C_VEL
LIN {X 0,Y 324.756,Z 400.028,A -85,B 0,C 180,E1 -15343.533,E2 -15343.533} C_VEL
LIN {X 0,Y 334.834,Z 415.409,A -85,B 0,C 180,E1 -15345.493,E2 -15345.493} C_VEL
LIN {X 0,Y 345.423,Z 433.68,A -85,B 0,C 180,E1 -15347.423,E2 -15347.423} C_VEL
LIN {X 0,Y 347.889,Z 438.395,A -85,B 0,C 180,E1 -15347.86,E2 -15347.86} C_VEL
LIN {X 0,Y 345.455,Z 513.037,A -85,B 0,C 180,E1 -15349.456,E2 -15349.456} C_VEL
LIN {X 0,Y 345.022,Z 530.432,A -85,B 0,C 180,E1 -15349.944,E2 -15349.944} C_VEL
LIN {X 0,Y 344.206,Z 544.89,A -85,B 0,C 180,E1 -15350.568,E2 -15350.568} C_VEL
LIN {X 0,Y 342.93,Z 558.782,A -85,B 0,C 180,E1 -15351.373,E2 -15351.373} C_VEL
LIN {X 0,Y 341.376,Z 572.553,A -85,B 0,C 180,E1 -15352.42,E2 -15352.42} C_VEL
LIN {X 0,Y 339.368,Z 586.128,A -85,B 0,C 180,E1 -15353.704,E2 -15353.704} C_VEL
LIN {X 0,Y 337.043,Z 598.947,A -85,B 0,C 180,E1 -15355.194,E2 -15355.194} C_VEL
LIN {X 0,Y 334.686,Z 610.917,A -85,B 0,C 180,E1 -15356.911,E2 -15356.911} C_VEL
LIN {X 0,Y 332.221,Z 621.756,A -85,B 0,C 180,E1 -15358.784,E2 -15358.784} C_VEL
LIN {X 0,Y 329.743,Z 631.86,A -85,B 0,C 180,E1 -15360.911,E2 -15360.911} C_VEL
LIN {X 0,Y 327.401,Z 640.765,A -85,B 0,C 180,E1 -15363.207,E2 -15363.207} C_VEL
LIN {X 0,Y 325.195,Z 648.712,A -85,B 0,C 180,E1 -15365.757,E2 -15365.757} C_VEL
LIN {X 0,Y 323.473,Z 654.975,A -85,B 0,C 180,E1 -15368.325,E2 -15368.325} C_VEL
LIN {X 0,Y 322.072,Z 659.772,A -85,B 0,C 180,E1 -15370.895,E2 -15370.895} C_VEL
LIN {X 0,Y 321.021,Z 663.247,A -85,B 0,C 180,E1 -15373.466,E2 -15373.466} C_VEL
LIN {X 0,Y 320.304,Z 665.508,A -85,B 0,C 180,E1 -15376.034,E2 -15376.034} C_VEL
LIN {X 0,Y 319.962,Z 666.609,A -85,B 0,C 180,E1 -15378.599,E2 -15378.599} C_VEL
LIN {X 0,Y 319.847,Z 666.504,A -85,B 0,C 180,E1 -15381.414,E2 -15381.414} C_VEL
LIN {X 0,Y 319.878,Z 665.403,A -85,B 0,C 180,E1 -15383.694,E2 -15383.694} C_VEL
LIN {X 0,Y 320.065,Z 663.167,A -85,B 0,C 180,E1 -15386.224,E2 -15386.224} C_VEL
LIN {X 0,Y 320.598,Z 659.763,A -85,B 0,C 180,E1 -15388.744,E2 -15388.744} C_VEL
LIN {X 0,Y 321.354,Z 655.143,A -85,B 0,C 180,E1 -15391.254,E2 -15391.254} C_VEL
LIN {X 0,Y 322.482,Z 649.164,A -85,B 0,C 180,E1 -15393.749,E2 -15393.749} C_VEL
LIN {X 0,Y 323.844,Z 641.676,A -85,B 0,C 180,E1 -15396.23,E2 -15396.23} C_VEL
LIN {X 0,Y 325.318,Z 633.703,A -85,B 0,C 180,E1 -15398.385,E2 -15398.385} C_VEL
LIN {X 0,Y 327.121,Z 624.098,A -85,B 0,C 180,E1 -15400.522,E2 -15400.522} C_VEL
LIN {X 0,Y 329.093,Z 612.492,A -85,B 0,C 180,E1 -15402.644,E2 -15402.644} C_VEL
LIN {X 0,Y 330.843,Z 600.494,A -85,B 0,C 180,E1 -15404.454,E2 -15404.454} C_VEL
LIN {X 0,Y 332.547,Z 588.465,A -85,B 0,C 180,E1 -15405.947,E2 -15405.947} C_VEL
LIN {X 0,Y 334.246,Z 575.293,A -85,B 0,C 180,E1 -15407.277,E2 -15407.277} C_VEL
LIN {X 0,Y 335.657,Z 561.675,A -85,B 0,C 180,E1 -15408.384,E2 -15408.384} C_VEL
LIN {X 0,Y 336.847,Z 546.441,A -85,B 0,C 180,E1 -15409.343,E2 -15409.343} C_VEL
LIN {X 0,Y 337.631,Z 531.036,A -85,B 0,C 180,E1 -15410.046,E2 -15410.046} C_VEL
LIN {X 0,Y 337.927,Z 516.122,A -85,B 0,C 180,E1 -15410.501,E2 -15410.501} C_VEL
LIN {X 0,Y 339.963,Z 431.831,A -85,B 0,C 180,E1 -15412.31,E2 -15412.31} C_VEL
LIN {X 0,Y 330.622,Z 412.452,A -85,B 0,C 180,E1 -15413.691,E2 -15413.691} C_VEL
LIN {X 0,Y 320.974,Z 394.748,A -85,B 0,C 180,E1 -15415.161,E2 -15415.161} C_VEL
LIN {X 0,Y 320.619,Z 394.243,A -85,B 0,C 180,E1 -15415.213,E2 -15415.213} C_VEL
LIN {X 0,Y 319.199,Z 392.681,A -85,B 0,C 180,E1 -15415.501,E2 -15415.501} C_VEL
LIN {X 0,Y 317.403,Z 391.711,A -85,B 0,C 180,E1 -15416.04,E2 -15416.04} C_VEL
LIN {X 0,Y 315.524,Z 391.807,A -85,B 0,C 180,E1 -15416.847,E2 -15416.847} C_VEL
LIN {X 0,Y 313.516,Z 392.178,A -85,B 0,C 180,E1 -15418.312,E2 -15418.312} C_VEL
LIN {X 0,Y 312.555,Z 392.201,A -85,B 0,C 180,E1 -15419.906,E2 -15419.906} C_VEL
LIN {X 0,Y 312.472,Z 392.171,A -85,B 0,C 180,E1 -15420.709,E2 -15420.709} C_VEL
LIN {X 0,Y 312.506,Z 392.179,A -85,B 0,C 180,E1 -15424.21,E2 -15424.21} C_VEL
LIN {X 0,Y 312.513,Z 392.179,A -85,B 0,C 180,E1 -15427.386,E2 -15427.386} C_VEL
LIN {X 0,Y 312.433,Z 392.186,A -85,B 0,C 180,E1 -15430.717,E2 -15430.717} C_VEL
LIN {X 0,Y 312.437,Z 392.186,A -85,B 0,C 180,E1 -15434.211,E2 -15434.211} C_VEL
LIN {X 0,Y 312.451,Z 392.184,A -85,B 0,C 180,E1 -15437.925,E2 -15437.925} C_VEL
LIN {X 0,Y 312.473,Z 392.18,A -85,B 0,C 180,E1 -15441.924,E2 -15441.924} C_VEL
LIN {X 0,Y 312.527,Z 392.181,A -85,B 0,C 180,E1 -15444.219,E2 -15444.219} C_VEL
LIN {X 0,Y 312.495,Z 392.181,A -85,B 0,C 180,E1 -15447.332,E2 -15447.332} C_VEL
LIN {X 0,Y 312.478,Z 392.179,A -85,B 0,C 180,E1 -15451.3,E2 -15451.3} C_VEL
LIN {X 0,Y 312.542,Z 392.178,A -85,B 0,C 180,E1 -15454.707,E2 -15454.707} C_VEL
LIN {X 0,Y 312.516,Z 392.182,A -85,B 0,C 180,E1 -15458.911,E2 -15458.911} C_VEL
LIN {X 0,Y 312.571,Z 392.172,A -85,B 0,C 180,E1 -15463.004,E2 -15463.004} C_VEL
LIN {X 0,Y 312.679,Z 392.151,A -85,B 0,C 180,E1 -15465.685,E2 -15465.685} C_VEL
LIN {X 0,Y 312.678,Z 392.113,A -85,B 0,C 180,E1 -15469.641,E2 -15469.641} C_VEL
LIN {X 0,Y 312.831,Z 392.139,A -85,B 0,C 180,E1 -15473.55,E2 -15473.55} C_VEL
LIN {X 0,Y 312.967,Z 392.113,A -85,B 0,C 180,E1 -15478.713,E2 -15478.713} C_VEL
LIN {X 0,Y 312.898,Z 392.127,A -85,B 0,C 180,E1 -15482.574,E2 -15482.574} C_VEL
LIN {X 0,Y 312.828,Z 392.14,A -85,B 0,C 180,E1 -15486.449,E2 -15486.449} C_VEL
LIN {X 0,Y 312.744,Z 392.142,A -85,B 0,C 180,E1 -15489.05,E2 -15489.05} C_VEL
LIN {X 0,Y 312.611,Z 392.168,A -85,B 0,C 180,E1 -15492.992,E2 -15492.992} C_VEL
LIN {X 0,Y 312.541,Z 392.175,A -85,B 0,C 180,E1 -15495.654,E2 -15495.654} C_VEL
LIN {X 0,Y 312.521,Z 392.176,A -85,B 0,C 180,E1 -15499.713,E2 -15499.713} C_VEL
LIN {X 0,Y 312.51,Z 392.175,A -85,B 0,C 180,E1 -15502.776,E2 -15502.776} C_VEL
LIN {X 0,Y 312.476,Z 392.182,A -85,B 0,C 180,E1 -15506.732,E2 -15506.732} C_VEL
LIN {X 0,Y 312.463,Z 392.186,A -85,B 0,C 180,E1 -15509.658,E2 -15509.658} C_VEL
LIN {X 0,Y 312.515,Z 392.166,A -85,B 0,C 180,E1 -15513.689,E2 -15513.689} C_VEL
LIN {X 0,Y 312.504,Z 392.178,A -85,B 0,C 180,E1 -15517.388,E2 -15517.388} C_VEL
LIN {X 0,Y 312.436,Z 392.193,A -85,B 0,C 180,E1 -15520.717,E2 -15520.717} C_VEL
LIN {X 0,Y 312.457,Z 392.186,A -85,B 0,C 180,E1 -15524.659,E2 -15524.659} C_VEL
LIN {X 0,Y 312.444,Z 392.231,A -85,B 0,C 180,E1 -15525.003,E2 -15525.003} C_VEL
LIN {X 0,Y 316.009,Z 403.797,A -85,B 0,C 180,E1 -15527.78,E2 -15527.78} C_VEL
LIN {X 0,Y 319.757,Z 417.249,A -85,B 0,C 180,E1 -15530.784,E2 -15530.784} C_VEL
LIN {X 0,Y 323.262,Z 431.561,A -85,B 0,C 180,E1 -15533.767,E2 -15533.767} C_VEL
LIN {X 0,Y 324.004,Z 435.441,A -85,B 0,C 180,E1 -15534.533,E2 -15534.533} C_VEL
LIN {X 0,Y 323.532,Z 439.575,A -85,B 0,C 180,E1 -15535.188,E2 -15535.188} C_VEL
LIN {X 0,Y 328.152,Z 474.622,A -85,B 0,C 180,E1 -15536.527,E2 -15536.527} C_VEL
LIN {X 0,Y 332.438,Z 511.726,A -85,B 0,C 180,E1 -15537.831,E2 -15537.831} C_VEL
LIN {X 0,Y 329.54,Z 608.583,A -85,B 0,C 180,E1 -15539.922,E2 -15539.922} C_VEL
LIN {X 0,Y 328.434,Z 624.282,A -85,B 0,C 180,E1 -15540.473,E2 -15540.473} C_VEL
LIN {X 0,Y 326.886,Z 639.403,A -85,B 0,C 180,E1 -15541.246,E2 -15541.246} C_VEL
LIN {X 0,Y 324.788,Z 654.537,A -85,B 0,C 180,E1 -15542.275,E2 -15542.275} C_VEL
LIN {X 0,Y 322.553,Z 669.216,A -85,B 0,C 180,E1 -15543.581,E2 -15543.581} C_VEL
LIN {X 0,Y 320.466,Z 682.22,A -85,B 0,C 180,E1 -15545.029,E2 -15545.029} C_VEL
LIN {X 0,Y 318.219,Z 694.9,A -85,B 0,C 180,E1 -15546.748,E2 -15546.748} C_VEL
LIN {X 0,Y 316.1,Z 707.37,A -85,B 0,C 180,E1 -15548.82,E2 -15548.82} C_VEL
LIN {X 0,Y 314.491,Z 717.054,A -85,B 0,C 180,E1 -15550.754,E2 -15550.754} C_VEL
LIN {X 0,Y 313.097,Z 726.587,A -85,B 0,C 180,E1 -15553.034,E2 -15553.034} C_VEL
LIN {X 0,Y 312.22,Z 734.919,A -85,B 0,C 180,E1 -15555.447,E2 -15555.447} C_VEL
LIN {X 0,Y 311.711,Z 741.14,A -85,B 0,C 180,E1 -15557.632,E2 -15557.632} C_VEL
LIN {X 0,Y 311.591,Z 747.222,A -85,B 0,C 180,E1 -15560.261,E2 -15560.261} C_VEL
LIN {X 0,Y 311.767,Z 751.588,A -85,B 0,C 180,E1 -15562.686,E2 -15562.686} C_VEL
LIN {X 0,Y 312.031,Z 754.459,A -85,B 0,C 180,E1 -15564.831,E2 -15564.831} C_VEL
LIN {X 0,Y 312.197,Z 756.727,A -85,B 0,C 180,E1 -15567.419,E2 -15567.419} C_VEL
LIN {X 0,Y 312.481,Z 757.42,A -85,B 0,C 180,E1 -15568.711,E2 -15568.711} C_VEL
LIN {X 0,Y 312.672,Z 757.792,A -85,B 0,C 180,E1 -15570,E2 -15570} C_VEL
LIN {X 0,Y 312.458,Z 757.802,A -85,B 0,C 180,E1 -15571.288,E2 -15571.288} C_VEL
LIN {X 0,Y 312.023,Z 756.903,A -85,B 0,C 180,E1 -15573.874,E2 -15573.874} C_VEL
LIN {X 0,Y 311.693,Z 754.747,A -85,B 0,C 180,E1 -15576.473,E2 -15576.473} C_VEL
LIN {X 0,Y 311.428,Z 751.361,A -85,B 0,C 180,E1 -15579.088,E2 -15579.088} C_VEL
LIN {X 0,Y 311.461,Z 746.716,A -85,B 0,C 180,E1 -15581.716,E2 -15581.716} C_VEL
LIN {X 0,Y 312.067,Z 740.471,A -85,B 0,C 180,E1 -15584.444,E2 -15584.444} C_VEL
LIN {X 0,Y 313.128,Z 733.267,A -85,B 0,C 180,E1 -15586.963,E2 -15586.963} C_VEL
LIN {X 0,Y 314.69,Z 725.407,A -85,B 0,C 180,E1 -15589.232,E2 -15589.232} C_VEL
LIN {X 0,Y 316.656,Z 716.326,A -85,B 0,C 180,E1 -15591.413,E2 -15591.413} C_VEL
LIN {X 0,Y 319.235,Z 704.847,A -85,B 0,C 180,E1 -15593.688,E2 -15593.688} C_VEL
LIN {X 0,Y 321.941,Z 693.455,A -85,B 0,C 180,E1 -15595.539,E2 -15595.539} C_VEL
LIN {X 0,Y 324.909,Z 680.753,A -85,B 0,C 180,E1 -15597.231,E2 -15597.231} C_VEL
LIN {X 0,Y 327.709,Z 667.465,A -85,B 0,C 180,E1 -15598.674,E2 -15598.674} C_VEL
LIN {X 0,Y 330.336,Z 654.206,A -85,B 0,C 180,E1 -15599.821,E2 -15599.821} C_VEL
LIN {X 0,Y 332.84,Z 639.78,A -85,B 0,C 180,E1 -15600.799,E2 -15600.799} C_VEL
LIN {X 0,Y 334.885,Z 624.953,A -85,B 0,C 180,E1 -15601.555,E2 -15601.555} C_VEL
LIN {X 0,Y 336.32,Z 609.748,A -85,B 0,C 180,E1 -15602.109,E2 -15602.109} C_VEL
LIN {X 0,Y 337.239,Z 589.653,A -85,B 0,C 180,E1 -15602.585,E2 -15602.585} C_VEL
LIN {X 0,Y 339.952,Z 512.164,A -85,B 0,C 180,E1 -15604.247,E2 -15604.247} C_VEL
LIN {X 0,Y 337.418,Z 489.325,A -85,B 0,C 180,E1 -15605.168,E2 -15605.168} C_VEL
LIN {X 0,Y 333.456,Z 462.006,A -85,B 0,C 180,E1 -15606.433,E2 -15606.433} C_VEL
LIN {X 0,Y 330.442,Z 444.886,A -85,B 0,C 180,E1 -15607.33,E2 -15607.33} C_VEL
LIN {X 0,Y 327.777,Z 439.219,A -85,B 0,C 180,E1 -15607.879,E2 -15607.879} C_VEL
LIN {X 0,Y 326.177,Z 435.483,A -85,B 0,C 180,E1 -15608.271,E2 -15608.271} C_VEL
LIN {X 0,Y 322.914,Z 423.363,A -85,B 0,C 180,E1 -15611.168,E2 -15611.168} C_VEL
LIN {X 0,Y 319.205,Z 411.312,A -85,B 0,C 180,E1 -15614.312,E2 -15614.312} C_VEL
LIN {X 0,Y 315.304,Z 400.062,A -85,B 0,C 180,E1 -15617.561,E2 -15617.561} C_VEL
LIN {X 0,Y 312.467,Z 392.189,A -85,B 0,C 180,E1 -15620.09,E2 -15620.09} C_VEL
LIN {X 0,Y 312.52,Z 392.177,A -85,B 0,C 180,E1 -15624.219,E2 -15624.219} C_VEL
LIN {X 0,Y 312.492,Z 392.183,A -85,B 0,C 180,E1 -15627.333,E2 -15627.333} C_VEL
LIN {X 0,Y 312.494,Z 392.188,A -85,B 0,C 180,E1 -15631.292,E2 -15631.292} C_VEL
LIN {X 0,Y 312.505,Z 392.184,A -85,B 0,C 180,E1 -15634.704,E2 -15634.704} C_VEL
LIN {X 0,Y 312.528,Z 392.184,A -85,B 0,C 180,E1 -15637.525,E2 -15637.525} C_VEL
LIN {X 0,Y 312.527,Z 392.181,A -85,B 0,C 180,E1 -15641.65,E2 -15641.65} C_VEL
LIN {X 0,Y 312.63,Z 392.163,A -85,B 0,C 180,E1 -15645.684,E2 -15645.684} C_VEL
LIN {X 0,Y 312.672,Z 392.155,A -85,B 0,C 180,E1 -15649.641,E2 -15649.641} C_VEL
LIN {X 0,Y 312.783,Z 392.149,A -85,B 0,C 180,E1 -15652.252,E2 -15652.252} C_VEL
LIN {X 0,Y 312.677,Z 392.16,A -85,B 0,C 180,E1 -15654.842,E2 -15654.842} C_VEL
LIN {X 0,Y 312.955,Z 392.125,A -85,B 0,C 180,E1 -15658.714,E2 -15658.714} C_VEL
LIN {X 0,Y 312.969,Z 392.116,A -85,B 0,C 180,E1 -15661.287,E2 -15661.287} C_VEL
LIN {X 0,Y 312.836,Z 392.105,A -85,B 0,C 180,E1 -15666.45,E2 -15666.45} C_VEL
LIN {X 0,Y 312.674,Z 392.16,A -85,B 0,C 180,E1 -15670.359,E2 -15670.359} C_VEL
LIN {X 0,Y 312.657,Z 392.133,A -85,B 0,C 180,E1 -15674.865,E2 -15674.865} C_VEL
LIN {X 0,Y 312.575,Z 392.162,A -85,B 0,C 180,E1 -15679.213,E2 -15679.213} C_VEL
LIN {X 0,Y 312.507,Z 392.173,A -85,B 0,C 180,E1 -15682.777,E2 -15682.777} C_VEL
LIN {X 0,Y 312.474,Z 392.164,A -85,B 0,C 180,E1 -15686.733,E2 -15686.733} C_VEL
LIN {X 0,Y 312.486,Z 392.189,A -85,B 0,C 180,E1 -15689.657,E2 -15689.657} C_VEL
LIN {X 0,Y 312.512,Z 392.18,A -85,B 0,C 180,E1 -15693.69,E2 -15693.69} C_VEL
LIN {X 0,Y 312.506,Z 392.172,A -85,B 0,C 180,E1 -15697.388,E2 -15697.388} C_VEL
LIN {X 0,Y 312.471,Z 392.291,A -85,B 0,C 180,E1 -15701.221,E2 -15701.221} C_VEL
LIN {X 0,Y 313.485,Z 395.065,A -85,B 0,C 180,E1 -15701.49,E2 -15701.49} C_VEL
LIN {X 0,Y 315.642,Z 397.674,A -85,B 0,C 180,E1 -15701.95,E2 -15701.95} C_VEL
LIN {X 0,Y 317.935,Z 401.067,A -85,B 0,C 180,E1 -15702.447,E2 -15702.447} C_VEL
LIN {X 0,Y 328.602,Z 417.21,A -85,B 0,C 180,E1 -15704.624,E2 -15704.624} C_VEL
LIN {X 0,Y 338.023,Z 433.203,A -85,B 0,C 180,E1 -15706.424,E2 -15706.424} C_VEL
LIN {X 0,Y 342.18,Z 440.817,A -85,B 0,C 180,E1 -15707.186,E2 -15707.186} C_VEL
LIN {X 0,Y 339.709,Z 513.777,A -85,B 0,C 180,E1 -15708.769,E2 -15708.769} C_VEL
LIN {X 0,Y 339.25,Z 531.274,A -85,B 0,C 180,E1 -15709.267,E2 -15709.267} C_VEL
LIN {X 0,Y 338.389,Z 545.789,A -85,B 0,C 180,E1 -15709.899,E2 -15709.899} C_VEL
LIN {X 0,Y 337.05,Z 559.907,A -85,B 0,C 180,E1 -15710.731,E2 -15710.731} C_VEL
LIN {X 0,Y 335.38,Z 573.947,A -85,B 0,C 180,E1 -15711.818,E2 -15711.818} C_VEL
LIN {X 0,Y 333.239,Z 587.838,A -85,B 0,C 180,E1 -15713.166,E2 -15713.166} C_VEL
LIN {X 0,Y 330.888,Z 600.217,A -85,B 0,C 180,E1 -15714.636,E2 -15714.636} C_VEL
LIN {X 0,Y 328.63,Z 611.17,A -85,B 0,C 180,E1 -15716.22,E2 -15716.22} C_VEL
LIN {X 0,Y 326.077,Z 622.138,A -85,B 0,C 180,E1 -15718.128,E2 -15718.128} C_VEL
LIN {X 0,Y 323.73,Z 631.342,A -85,B 0,C 180,E1 -15720.047,E2 -15720.047} C_VEL
LIN {X 0,Y 321.255,Z 640.257,A -85,B 0,C 180,E1 -15722.299,E2 -15722.299} C_VEL
LIN {X 0,Y 319.034,Z 648.129,A -85,B 0,C 180,E1 -15724.765,E2 -15724.765} C_VEL
LIN {X 0,Y 317.211,Z 654.317,A -85,B 0,C 180,E1 -15727.188,E2 -15727.188} C_VEL
LIN {X 0,Y 315.636,Z 659.525,A -85,B 0,C 180,E1 -15729.812,E2 -15729.812} C_VEL
LIN {X 0,Y 314.676,Z 662.517,A -85,B 0,C 180,E1 -15731.78,E2 -15731.78} C_VEL
LIN {X 0,Y 313.752,Z 665.435,A -85,B 0,C 180,E1 -15734.408,E2 -15734.408} C_VEL
LIN {X 0,Y 313.125,Z 667.175,A -85,B 0,C 180,E1 -15737.03,E2 -15737.03} C_VEL
LIN {X 0,Y 312.873,Z 667.725,A -85,B 0,C 180,E1 -15739.648,E2 -15739.648} C_VEL
LIN {X 0,Y 312.841,Z 667.174,A -85,B 0,C 180,E1 -15742.254,E2 -15742.254} C_VEL
LIN {X 0,Y 312.821,Z 665.566,A -85,B 0,C 180,E1 -15744.845,E2 -15744.845} C_VEL
LIN {X 0,Y 313.304,Z 662.797,A -85,B 0,C 180,E1 -15747.429,E2 -15747.429} C_VEL
LIN {X 0,Y 313.944,Z 658.864,A -85,B 0,C 180,E1 -15750,E2 -15750} C_VEL
LIN {X 0,Y 314.895,Z 653.651,A -85,B 0,C 180,E1 -15752.559,E2 -15752.559} C_VEL
LIN {X 0,Y 316.172,Z 647.017,A -85,B 0,C 180,E1 -15755.101,E2 -15755.101} C_VEL
LIN {X 0,Y 317.722,Z 638.775,A -85,B 0,C 180,E1 -15757.627,E2 -15757.627} C_VEL
LIN {X 0,Y 319.455,Z 629.994,A -85,B 0,C 180,E1 -15759.817,E2 -15759.817} C_VEL
LIN {X 0,Y 321.419,Z 619.426,A -85,B 0,C 180,E1 -15761.989,E2 -15761.989} C_VEL
LIN {X 0,Y 323.26,Z 608.58,A -85,B 0,C 180,E1 -15763.837,E2 -15763.837} C_VEL
LIN {X 0,Y 324.932,Z 596.737,A -85,B 0,C 180,E1 -15765.525,E2 -15765.525} C_VEL
LIN {X 0,Y 326.899,Z 583.628,A -85,B 0,C 180,E1 -15767.033,E2 -15767.033} C_VEL
LIN {X 0,Y 328.359,Z 570.824,A -85,B 0,C 180,E1 -15768.242,E2 -15768.242} C_VEL
LIN {X 0,Y 329.75,Z 556.805,A -85,B 0,C 180,E1 -15769.29,E2 -15769.29} C_VEL
LIN {X 0,Y 330.833,Z 541.908,A -85,B 0,C 180,E1 -15770.141,E2 -15770.141} C_VEL
LIN {X 0,Y 331.404,Z 526.967,A -85,B 0,C 180,E1 -15770.758,E2 -15770.758} C_VEL
LIN {X 0,Y 331.87,Z 503.419,A -85,B 0,C 180,E1 -15771.347,E2 -15771.347} C_VEL
LIN {X 0,Y 333.782,Z 434.034,A -85,B 0,C 180,E1 -15772.847,E2 -15772.847} C_VEL
LIN {X 0,Y 324.793,Z 415.357,A -85,B 0,C 180,E1 -15774.221,E2 -15774.221} C_VEL
LIN {X 0,Y 315.755,Z 398.808,A -85,B 0,C 180,E1 -15775.641,E2 -15775.641} C_VEL
LIN {X 0,Y 312.79,Z 393.488,A -85,B 0,C 180,E1 -15776.127,E2 -15776.127} C_VEL
LIN {X 0,Y 312.499,Z 392.185,A -85,B 0,C 180,E1 -15776.22,E2 -15776.22} C_VEL
LIN {X 0,Y 312.466,Z 392.17,A -85,B 0,C 180,E1 -15779.658,E2 -15779.658} C_VEL
LIN {X 0,Y 312.472,Z 392.171,A -85,B 0,C 180,E1 -15780.709,E2 -15780.709} C_VEL
LIN {X 0,Y 311.858,Z 392.263,A -85,B 0,C 180,E1 -15781.785,E2 -15781.785} C_VEL
LIN {X 0,Y 309.042,Z 392.615,A -85,B 0,C 180,E1 -15783.537,E2 -15783.537} C_VEL
LIN {X 0,Y 306.613,Z 392.918,A -85,B 0,C 180,E1 -15784.958,E2 -15784.958} C_VEL
LIN {X 0,Y 305.553,Z 393.048,A -85,B 0,C 180,E1 -15786.058,E2 -15786.058} C_VEL
LIN {X 0,Y 305.459,Z 393.057,A -85,B 0,C 180,E1 -15786.431,E2 -15786.431} C_VEL
LIN {X 0,Y 305.407,Z 393.059,A -85,B 0,C 180,E1 -15790.115,E2 -15790.115} C_VEL
LIN {X 0,Y 305.401,Z 393.061,A -85,B 0,C 180,E1 -15793.659,E2 -15793.659} C_VEL
LIN {X 0,Y 305.431,Z 393.058,A -85,B 0,C 180,E1 -15797.418,E2 -15797.418} C_VEL
LIN {X 0,Y 305.441,Z 393.056,A -85,B 0,C 180,E1 -15801.592,E2 -15801.592} C_VEL
LIN {X 0,Y 305.458,Z 393.062,A -85,B 0,C 180,E1 -15804.886,E2 -15804.886} C_VEL
LIN {X 0,Y 305.435,Z 393.064,A -85,B 0,C 180,E1 -15808.359,E2 -15808.359} C_VEL
LIN {X 0,Y 305.441,Z 393.061,A -85,B 0,C 180,E1 -15812.6,E2 -15812.6} C_VEL
LIN {X 0,Y 305.469,Z 393.05,A -85,B 0,C 180,E1 -15815.535,E2 -15815.535} C_VEL
LIN {X 0,Y 305.477,Z 393.053,A -85,B 0,C 180,E1 -15819.812,E2 -15819.812} C_VEL
LIN {X 0,Y 305.545,Z 393.049,A -85,B 0,C 180,E1 -15823.977,E2 -15823.977} C_VEL
LIN {X 0,Y 305.578,Z 393.024,A -85,B 0,C 180,E1 -15826.703,E2 -15826.703} C_VEL
LIN {X 0,Y 305.714,Z 392.999,A -85,B 0,C 180,E1 -15831.302,E2 -15831.302} C_VEL
LIN {X 0,Y 305.777,Z 393.016,A -85,B 0,C 180,E1 -15833.401,E2 -15833.401} C_VEL
LIN {X 0,Y 305.933,Z 392.989,A -85,B 0,C 180,E1 -15838.683,E2 -15838.683} C_VEL
LIN {X 0,Y 305.928,Z 393.003,A -85,B 0,C 180,E1 -15841.316,E2 -15841.316} C_VEL
LIN {X 0,Y 305.649,Z 393.029,A -85,B 0,C 180,E1 -15845.277,E2 -15845.277} C_VEL
LIN {X 0,Y 305.736,Z 393.019,A -85,B 0,C 180,E1 -15847.927,E2 -15847.927} C_VEL
LIN {X 0,Y 305.585,Z 393.045,A -85,B 0,C 180,E1 -15851.946,E2 -15851.946} C_VEL
LIN {X 0,Y 305.545,Z 393.041,A -85,B 0,C 180,E1 -15854.973,E2 -15854.973} C_VEL
LIN {X 0,Y 305.492,Z 393.048,A -85,B 0,C 180,E1 -15858.788,E2 -15858.788} C_VEL
LIN {X 0,Y 305.45,Z 393.054,A -85,B 0,C 180,E1 -15863.026,E2 -15863.026} C_VEL
LIN {X 0,Y 305.444,Z 393.057,A -85,B 0,C 180,E1 -15866.189,E2 -15866.189} C_VEL
LIN {X 0,Y 305.419,Z 393.064,A -85,B 0,C 180,E1 -15869.025,E2 -15869.025} C_VEL
LIN {X 0,Y 305.431,Z 393.061,A -85,B 0,C 180,E1 -15871.953,E2 -15871.953} C_VEL
LIN {X 0,Y 305.456,Z 393.055,A -85,B 0,C 180,E1 -15875.114,E2 -15875.114} C_VEL
LIN {X 0,Y 305.429,Z 393.051,A -85,B 0,C 180,E1 -15878.525,E2 -15878.525} C_VEL
LIN {X 0,Y 305.429,Z 393.053,A -85,B 0,C 180,E1 -15882.581,E2 -15882.581} C_VEL
LIN {X 0,Y 305.44,Z 393.218,A -85,B 0,C 180,E1 -15884.312,E2 -15884.312} C_VEL
LIN {X 0,Y 309.02,Z 404.753,A -85,B 0,C 180,E1 -15887.176,E2 -15887.176} C_VEL
